// TIA Portal project "FillerMachine" (V15)
// Maquina llenadora Fuente Pura CCN

(* hardware
DEVICE "ET 200SP station_1"  ET 200SP-Station
   slot 0: "Rack_0"  Rack  6ES5 710-8MAx1
   slot 1: "PLC_1"  CPU 1510SP-1 PN  6ES7 510-1DJ01-0AB0  V2.5
   slot 2: "DI 8x24VDC ST_1"  DI 8x24VDC ST  6ES7 131-6BF00-0BA0  V1.1
      slot 1: "DI 8x24VDC ST_1"  DI 8x24VDC ST
   slot 3: "DI 8x24VDC ST_2"  DI 8x24VDC ST  6ES7 131-6BF01-0BA0  V0.0
      slot 1: "DI 8x24VDC ST_2"  DI 8x24VDC ST
   slot 4: "DI 8x24VDC ST_3"  DI 8x24VDC ST  6ES7 131-6BF01-0BA0  V0.0
      slot 1: "DI 8x24VDC ST_3"  DI 8x24VDC ST
   slot 5: "DQ 8x24VDC/0.5A ST_1"  DQ 8x24VDC/0.5A ST  6ES7 132-6BF01-0BA0  V0.0
      slot 1: "DQ 8x24VDC/0.5A ST_1"  DQ 8x24VDC/0.5A ST
   slot 6: "DQ 8x24VDC/0.5A ST_2"  DQ 8x24VDC/0.5A ST  6ES7 132-6BF01-0BA0  V0.0
      slot 1: "DQ 8x24VDC/0.5A ST_2"  DQ 8x24VDC/0.5A ST
   slot 7: "DQ 8x24VDC/0.5A ST_3"  DQ 8x24VDC/0.5A ST  6ES7 132-6BF01-0BA0  V0.0
      slot 1: "DQ 8x24VDC/0.5A ST_3"  DQ 8x24VDC/0.5A ST
   slot 8: "Server module_1"  Server module  6ES7 193-6PA00-0AA0  V1.1
      slot 1: "Server module_1"  Server module
   slot 127: "BA 2xRJ45"  BA 2xRJ45  6ES7 193-6AR00-0AA0  V0.0
      slot 32769: "Port_1"  6ES7 193-6AR00-0AA0
      slot 32770: "Port_2"  6ES7 193-6AR00-0AA0
DEVICE "HMI_1"  KTP600 Basic color PN
   slot 0: "HMI_1"  KTP600 Basic color PN  6AV6 647-0AD11-3AX0  12.0.0.0
   slot 1: "HMI_RT_2"  KTP600 Basic color PN  6AV6 647-0AD11-3AX0  12.0.0.0
   slot 5: "HMI_1.IE_CP_1"  PROFINET Interface  12.0.0.0
      slot 1: "PROFINET Interface_1"  PROFINET Interface
         slot 1: "Port_1"  Port
*)

// ===== PLC "PLC_1"  CPU 1510SP-1 PN =====

VAR_GLOBAL   // PLC tag table "Default tag table"
   "E_Stop" AT %I0.0 : Bool;
   "F_TriggerPump" AT %I0.1 : Bool;
   "ACKPump" AT %I0.2 : Bool;
   "F_TriggerClamp" AT %I0.3 : Bool;
   "ACKTap" AT %I0.4 : Bool;
   "F_TriggerTransp1" AT %I0.5 : Bool;
   "ACKTransp1" AT %I0.6 : Bool;
   "F_TriggerTransp2" AT %I0.7 : Bool;
   "ACKTransp2" AT %I1.0 : Bool;
   "S_ConvellorClearence_In" AT %I1.1 : Bool;
   "S_InBottle" AT %I1.2 : Bool;
   "S_OutBottle" AT %I1.6 : Bool;
   "S_LastBottle" AT %I1.4 : Bool;
   "S_Bottle_Convellor1" AT %I1.5 : Bool;
   "S_LevelH" AT %I1.3 : Bool;
   "S_LevelL" AT %I1.7 : Bool;
   "S_BottleTap" AT %I2.0 : Bool;
   "S_TranspClamp" AT %I2.1 : Bool;
   "PumpVLow" AT %Q0.0 : Bool;
   "PumpVHigh" AT %Q0.1 : Bool;
   "PumpStop" AT %Q0.2 : Bool;
   "MotorTap" AT %Q0.3 : Bool;
   "MotorTrans1" AT %Q0.4 : Bool;
   "MotorTrans2" AT %Q0.5 : Bool;
   "EVPrincip" AT %Q1.6 : Bool;
   "EVBlowCylindIN" AT %Q1.7 : Bool;
   "EVCylindBottleHigh" AT %Q2.0 : Bool;
   "EVCylindNeck" AT %Q2.1 : Bool;
   "EVDoorIn" AT %Q2.2 : Bool;
   "EVDoorOut" AT %Q2.3 : Bool;
   "EVClampBotNeck" AT %Q2.4 : Bool;
   "EVClampDoor" AT %Q2.5 : Bool;
   "EVSuperClamp" AT %Q2.6 : Bool;
   "EVMandrilcylindUpDown" AT %Q2.7 : Bool;
   "Start_hmi" AT %M11.0 : Bool;
   "MBandaT-On" AT %M10.1 : Bool;
   "MFillScreen" AT %M10.2 : Bool;
   "MBottleProcess" AT %MD100 : DInt;
   "MBottleCounterIN" AT %MD108 : DInt;
   "MBottleCounterOut" AT %MD128 : DInt;
   "MEnableClampValve" AT %MD132 : DInt;
   "MFillFinish" AT %M10.3 : Bool;
   "M_stop_hmi" AT %M11.1 : Bool;
   "S_ConvellorClearence_bit" AT %M20.3 : Bool;
   "S_InBottle_bit" AT %M20.4 : Bool;
   "S_OutBottle_bit" AT %M20.5 : Bool;
   "S_LastBottle_bit" AT %M20.6 : Bool;
   "S_Bottle_Convellor1_bit" AT %M20.7 : Bool;
   "S_LevelH_bit" AT %M21.0 : Bool;
   "S_LevelL_bit" AT %M21.1 : Bool;
   "S_BottleTap_bit" AT %M21.2 : Bool;
   "S_TranspClamp_bit" AT %M21.3 : Bool;
   "PumpVLow_bit" AT %M21.4 : Bool;
   "PumpVHigh_bit" AT %M21.5 : Bool;
   "PumpStop_bit" AT %M21.6 : Bool;
   "MotorTap_bit" AT %M21.7 : Bool;
   "MotorTrans1_bit" AT %M22.0 : Bool;
   "MotorTrans2_bit" AT %M22.1 : Bool;
   "EVPrincip_bit" AT %M22.2 : Bool;
   "EVBlowCylindIN_bit" AT %M22.3 : Bool;
   "EVMandrilcylindUpDown_bit" AT %M22.4 : Bool;
   "EVCylindNeck_bit" AT %M22.5 : Bool;
   "EVDoorIn_bit" AT %M50.1 : Bool;
   "EVDoorOut_bit" AT %M22.7 : Bool;
   "EVClampBotNeck_bit" AT %M23.0 : Bool;
   "EVClampDoor_bit" AT %M23.1 : Bool;
   "EVSuperClamp_bit" AT %M23.2 : Bool;
   "Alarm" AT %M24.0 : Bool;
   "F_TriggerPump_bit" AT %M24.1 : Bool;
   "F_TriggerClamp_bit" AT %M24.3 : Bool;
   "F_TriggerTransp1_bit" AT %M24.5 : Bool;
   "F_TriggerTransp2_bit" AT %M24.7 : Bool;
   "Run" AT %M25.1 : Bool;
   "Stop_bit" AT %M25.2 : Bool;
   "StageLL0" AT %M25.3 : Bool;
   "StageLL1" AT %M25.4 : Bool;
   "MBottleCounterR" AT %M25.5 : Bool;
   "ProcessFillingTimeR" AT %M25.6 : Bool;
   "StageLL2" AT %M25.7 : Bool;
   "MBottleclampRt" AT %M27.3 : Bool;
   "E_Trans1_hmi" AT %M27.4 : Bool;
   "E_Trans2_hmi" AT %M27.5 : Bool;
   "Pump_hmi" AT %M27.6 : Bool;
   "E_MotorTap_hmi" AT %M27.7 : Bool;
   "EVCylindBottleHigh_bit" AT %M28.0 : Bool;
   "StageLL3" AT %M28.1 : Bool;
   "StageLL4" AT %M28.2 : Bool;
   "StageLL5" AT %M28.3 : Bool;
   "StageLL6" AT %M28.4 : Bool;
   "StageLL7" AT %M28.5 : Bool;
   "StageLL8" AT %M28.6 : Bool;
   "StageLL9" AT %M28.7 : Bool;
   "StageLL10" AT %M29.0 : Bool;
   "StageLL11" AT %M29.1 : Bool;
   "Tag_1" AT %M400.1 : Bool;
   "StageLL12" AT %M29.2 : Bool;
   "StageLL13" AT %M29.3 : Bool;
   "StageLL14" AT %M29.4 : Bool;
   "Tag_2" AT %M400.2 : Bool;
   "StageLL00" AT %M29.5 : Bool;
   "MBottleCounterOutR" AT %M29.6 : Bool;
   "StageTap0" AT %M29.7 : Bool;
   "StageTap1" AT %M30.0 : Bool;
   "StageTap2" AT %M30.1 : Bool;
   "StageTap3" AT %M30.2 : Bool;
   "StageTap4" AT %M30.3 : Bool;
   "StageTap5" AT %M30.4 : Bool;
   "MTapProcessR" AT %M30.5 : Bool;
   "StageCon0" AT %M30.6 : Bool;
   "StageCon1" AT %M30.7 : Bool;
   "StageCon2" AT %M31.0 : Bool;
   "StageCon3" AT %M31.1 : Bool;
   "Timer1R" AT %M31.2 : Bool;
   "MConvT2R" AT %M31.3 : Bool;
   "StageCon4" AT %M31.4 : Bool;
   "E_stop_bit" AT %M31.5 : Bool;
   "ACKTap_bit" AT %M32.0 : Bool;
   "ACKPump_bit" AT %M32.1 : Bool;
   "ACKTransp1_bit" AT %M32.2 : Bool;
   "ACKTransp2_bit" AT %M32.3 : Bool;
   "MotorTap_fail" AT %M32.4 : Bool;
   "System_Byte" AT %MB1 : Byte;
   "RebuildMachine" AT %M1.0 : Bool;
   "DiagStatusUpdate" AT %M1.1 : Bool;
   "AlwaysTRUE" AT %M1.2 : Bool;
   "AlwaysFALSE" AT %M1.3 : Bool;
   "Clock_Byte" AT %MB0 : Byte;
   "Clock_10Hz" AT %M0.0 : Bool;
   "Clock_5Hz" AT %M0.1 : Bool;
   "Clock_2.5Hz" AT %M0.2 : Bool;
   "Clock_2Hz" AT %M0.3 : Bool;
   "Clock_1.25Hz" AT %M0.4 : Bool;
   "Clock_1Hz" AT %M0.5 : Bool;
   "Clock_0.625Hz" AT %M0.6 : Bool;
   "Clock_0.5Hz" AT %M0.7 : Bool;
   "MotorTransp1_fail" AT %M32.5 : Bool;
   "MotorTransp2_fail" AT %M32.6 : Bool;
   "MotorPump_fail" AT %M32.7 : Bool;
   "E_Manual" AT %M33.0 : Bool;
   "TimeFilling_hmi" AT %MD124 : Real;
   "TimeFilling_high" AT %MD104 : Real;
   "TimeFilling_low" AT %MD112 : Real;
   "TimeFilling_highT" AT %MD116 : Time;
   "TimeFilling_lowT" AT %MD120 : Time;
   "TimeFilling_highD" AT %MD54 : DInt;
   "TimeFilling_lowD" AT %MD58 : DInt;
   "TimeFilling_highPer" AT %MD62 : Real;
   "TimeFilling_lowPer" AT %MD66 : Real;
   "M_Stop" AT %M37.2 : Bool;
   "M_Stop_Counter_R" AT %M37.0 : Bool;
   "Stop_Batch" AT %M37.1 : Bool;
   "TapPPM" AT %MW4 : Word;
   "ResetTapPPM" AT %M37.3 : Bool;
   "ONS1" AT %M37.4 : Bool;
   "TapPPM_HMI" AT %MW6 : Word;
   "EstimatePPM_HMI" AT %MD70 : Real;
   "PumpVLow_hmi" AT %M37.5 : Bool;
   "EVBlowCylindIN_hmi" AT %M37.6 : Bool;
   "EVCylindBottleHigh_hmi" AT %M37.7 : Bool;
   "EVCylindNeck_hmi" AT %M39.0 : Bool;
   "EVPrincip_hmi" AT %M39.1 : Bool;
   "EVDoorIn_hmi" AT %M50.0 : Bool;
   "EVDoorOut_hmi" AT %M39.3 : Bool;
   "EVClampBotNeck_hmi" AT %M39.4 : Bool;
   "EVClampDoor_hmi" AT %M39.5 : Bool;
   "EVSuperClamp_hmi" AT %M50.2 : Bool;
   "EVMandrilcylindUpDown_hmi" AT %M50.3 : Bool;
   "E_Manual_hmi" AT %M31.6 : Bool;
   "Tag_3" AT %I2.4 : Bool;
   "Tag_4" AT %I2.3 : Bool;
   "Tag_5" AT %M24.2 : Bool;
   "Tag_6" AT %M140.1 : Bool;
   "Tag_7" AT %MD150 : DInt;
   "Tag_8" AT %MD154 : DInt;
   "Tag_9" AT %MD158 : DInt;
   "Tag_10" AT %MD162 : DInt;
   "Tag_11" AT %MD166 : DInt;
   "Tag_12" AT %MD170 : DInt;
   "Tag_13" AT %MD172 : DInt;
   "Tag_14" AT %MD176 : DInt;
   "Tag_15" AT %MD180 : DInt;
   "Tag_16" AT %MD184 : DInt;
   "Tag_17" AT %MD188 : Real;
   "Tag_18" AT %MD192 : Real;
   "Tag_19" AT %MD200 : Real;
   "Tag_20" AT %MD204 : Real;
   "Tag_21" AT %MD208 : Real;
   "Tag_22" AT %MD212 : Real;
   "Tag_23" AT %MD216 : Real;
   "Tag_24" AT %MD220 : Real;
   "Tag_25" AT %MD224 : Real;
   "Tag_26" AT %MD228 : Real;
   "Tag_27" AT %MD232 : Real;
   "Tag_28" AT %MD236 : Real;
   "R_time_b_neck" AT %M40.0 : Bool;
   "P_sensor_out" AT %M40.1 : Bool;
   "Tag_30" AT %MD240 : Real;
   "Tag_31" AT %MD244 : DInt;
   "PumpVHihg_hmi" AT %M40.2 : Bool;
   "Tag_32" AT %MD248 : Real;
   "Tag_33" AT %MD252 : DInt;
   "Tag_34" AT %MD256 : Real;
   "Tag_35" AT %MD260 : DInt;
   "P_Stop_hmi" AT %M40.4 : Bool;
   "Stop_hmi" AT %M40.5 : Bool;
   "WashProcess_1" AT %M10.4 : Bool;
   "WashProcess_hmi" AT %M10.5 : Bool;
   "RunWash" AT %M10.6 : Bool;
   "RWashProcess" AT %M10.7 : Bool;
   "Tag_36" AT %MD264 : Real;
   "Tag_37" AT %MD268 : DInt;
   "ValueProduction" AT %MD272 : DWord;
   "RProduction" AT %M31.7 : Bool;
   "Tag_29" AT %MD276 : Real;
   "Tag_38" AT %MD280 : DInt;
   "WashProcess_2" AT %M11.3 : Bool;
   "WashProcess_3" AT %M11.4 : Bool;
   "WashProcess_0" AT %M11.5 : Bool;
   "WashProcess_4" AT %M11.6 : Bool;
   "ret_val_RD_LOC" AT %MW284 : Int;
   "ret_val_RD_SYS" AT %MW288 : Int;
   "ret_val_WR_SYS" AT %MW292 : Int;
   "write_time" AT %M140.2 : Bool;
   "write_time_p" AT %M140.3 : Bool;
   "RestValve" AT %Q0.6 : Bool;
   "RestValve_bit" AT %M140.4 : Bool;
END_VAR

DATA_BLOCK "MotorTap_DB"   // DB1
{ S7_Optimized_Access := 'TRUE' }
VERSION : 0.1
// stored: InstanceOfName MotorData
"MotorData"
BEGIN
END_DATA_BLOCK

DATA_BLOCK "MotorTransp1_DB"   // DB5
{ S7_Optimized_Access := 'TRUE' }
VERSION : 0.1
// stored: InstanceOfName MotorData
"MotorData"
BEGIN
END_DATA_BLOCK

DATA_BLOCK "MotorTransp1"   // DB7
{ S7_Optimized_Access := 'TRUE' }
VERSION : 0.1
// stored: InstanceOfName MotorData
"MotorData"
BEGIN
END_DATA_BLOCK

DATA_BLOCK "MotorTransp2_DB"   // DB8
{ S7_Optimized_Access := 'TRUE' }
VERSION : 0.1
// stored: InstanceOfName MotorData
"MotorData"
BEGIN
END_DATA_BLOCK

DATA_BLOCK "init_var"   // DB9
{ S7_Optimized_Access := 'TRUE' }
VERSION : 0.1
   VAR RETAIN
      fillNo : Int := 8;
      filltime : Real := 9.0;
      fillPerHigh : Real := 70.0;
      fillPerLow : Real := 30.0;
   END_VAR
   VAR
      TimeConveyorBatch : Time := T#8.0S;
      TimeBeforeCylNeck : Time := T#0.5S;
      TimeCylNeck : Time := T#2S;
      TimeCylBottleHigh : Time := T#2S;
      TimeResetVLow : Time := T#2S;
      TimeRCyl_Neck_BottleHigh : Time := T#2S;
      TimeLastBottleOut : Time := T#2S;
      TimeClamp_Door_Neck : Time := T#2S;
      TimeClamp_Mandril : Time := T#2S;
      TimeSuperClamp : Time := T#0.05S;
   END_VAR
   VAR RETAIN
      RTimeConveyorBatch : Real := 2.0;
      RTimeBeforeCylNeck : Real := 0.5;
      RTimeCylBottleHigh : Real := 0.5;
      RTimeResetVLow : Real := 0.5;
      RTimeClamp_Door_Neck : Real := 0.5;
      RTimeClamp_Mandril : Real := 0.04;
      RTimeCylNeck : Real := 0.5;
      RTimeSuperClamp : Real := 2.0;
      RTimeRCyl_Neck_BottleHigh : Real := 1.0;
      RTimeRMandril_SuperClamp : Real := 2.0;
      RTimeLastBottleOut : Real := 0.5;
   END_VAR
   VAR
      TimeRMandril_SuperClamp : Time;
      TimeBNeck : Time;
   END_VAR
   VAR RETAIN
      RTimeBNeck : Real := 0.15;
      ROnDelayCylIn : Real := 0.5;
   END_VAR
   VAR
      TOnDelayCylIn : Time := T#0.5S;
   END_VAR
   VAR RETAIN
      ROnDelayDoorIn : Real := 0.9;
   END_VAR
   VAR
      TOnDelayDoorIn : Time := T#0.9S;
   END_VAR
   VAR RETAIN
      ROnDelayNeckClamp : Real := 0.5;
   END_VAR
   VAR
      TOnDelayNeckClamp : Time := T#0.5S;
      TWashTime : Time := T#120S;
   END_VAR
   VAR RETAIN
      RWashTime : Real := 120.0;
   END_VAR
BEGIN
END_DATA_BLOCK

DATA_BLOCK "DB_Alarms"   // DB13
{ S7_Optimized_Access := 'FALSE' }
VERSION : 0.1
   VAR
      E_Stop_alm : Bool;
      T_Pump_alm : Bool;
      T_Transp1_alm : Bool;
      T_Transp2_alm : Bool;
      T_Clamp_alm_1 : Bool;
      alarms_active : Bool;
   END_VAR
BEGIN
END_DATA_BLOCK

DATA_BLOCK "DB_Time"   // DB19
{ S7_Optimized_Access := 'TRUE' }
VERSION : 0.1
   VAR
      time_local_Read : DTL;
      time_system_WRITE : DTL;
   END_VAR
BEGIN
END_DATA_BLOCK

// folder: System blocks/Program resources

DATA_BLOCK "TimerStage2"   // DB2
{ S7_Optimized_Access := 'TRUE' }
AUTHOR : Simatic
FAMILY : IEC
NAME : IEC_TMR
VERSION : 1.0
// stored: InstanceOfName IEC_TIMER
"IEC_TIMER"
BEGIN
END_DATA_BLOCK

DATA_BLOCK "Timer_Cyl_Out"   // DB3
{ S7_Optimized_Access := 'TRUE' }
AUTHOR : Simatic
FAMILY : IEC
NAME : IEC_TMR
VERSION : 1.0
// stored: InstanceOfName IEC_TIMER
"IEC_TIMER"
BEGIN
END_DATA_BLOCK

DATA_BLOCK "TimeNeckWash"   // DB4
{ S7_Optimized_Access := 'TRUE' }
AUTHOR : Simatic
FAMILY : IEC
NAME : IEC_TMR
VERSION : 1.0
// stored: InstanceOfName IEC_TIMER
"IEC_TIMER"
BEGIN
END_DATA_BLOCK

DATA_BLOCK "IEC_Timer_0_DB_4"   // DB6
{ S7_Optimized_Access := 'TRUE' }
AUTHOR : Simatic
FAMILY : IEC
NAME : IEC_TMR
VERSION : 1.0
// stored: InstanceOfName IEC_TIMER
"IEC_TIMER"
BEGIN
END_DATA_BLOCK

DATA_BLOCK "CounterTapPPM"   // DB10
{ S7_Optimized_Access := 'TRUE' }
AUTHOR : Simatic
FAMILY : IEC
NAME : CNTR
VERSION : 1.0
// stored: InstanceOfName IEC_COUNTER
"IEC_COUNTER"
BEGIN
END_DATA_BLOCK

DATA_BLOCK "CounterTap"   // DB11
{ S7_Optimized_Access := 'TRUE' }
AUTHOR : Simatic
FAMILY : IEC
NAME : CNTR
VERSION : 1.0
// stored: InstanceOfName IEC_COUNTER
"IEC_COUNTER"
BEGIN
END_DATA_BLOCK

DATA_BLOCK "Delay_door_in"   // DB12
{ S7_Optimized_Access := 'TRUE' }
AUTHOR : Simatic
FAMILY : IEC
NAME : IEC_TMR
VERSION : 1.0
// stored: InstanceOfName IEC_TIMER
"IEC_TIMER"
BEGIN
END_DATA_BLOCK

DATA_BLOCK "TimerPPMDisable"   // DB14
{ S7_Optimized_Access := 'TRUE' }
AUTHOR : Simatic
FAMILY : IEC
NAME : IEC_TMR
VERSION : 1.0
// stored: InstanceOfName IEC_TIMER
"IEC_TIMER"
BEGIN
END_DATA_BLOCK

DATA_BLOCK "IEC_Timer_0_DB"   // DB15
{ S7_Optimized_Access := 'TRUE' }
AUTHOR : Simatic
FAMILY : IEC
NAME : IEC_TMR
VERSION : 1.0
// stored: InstanceOfName IEC_TIMER
"IEC_TIMER"
BEGIN
END_DATA_BLOCK

DATA_BLOCK "TimerStageWash"   // DB16
{ S7_Optimized_Access := 'TRUE' }
AUTHOR : Simatic
FAMILY : IEC
NAME : IEC_TMR
VERSION : 1.0
// stored: InstanceOfName IEC_TIMER
"IEC_TIMER"
BEGIN
END_DATA_BLOCK

DATA_BLOCK "TimeValvWash"   // DB17
{ S7_Optimized_Access := 'TRUE' }
AUTHOR : Simatic
FAMILY : IEC
NAME : IEC_TMR
VERSION : 1.0
// stored: InstanceOfName IEC_TIMER
"IEC_TIMER"
BEGIN
END_DATA_BLOCK

DATA_BLOCK "CounterProduction"   // DB18
{ S7_Optimized_Access := 'TRUE' }
AUTHOR : Simatic
FAMILY : IEC
NAME : CNTR
VERSION : 1.0
// stored: InstanceOfName IEC_COUNTER
"IEC_COUNTER"
BEGIN
END_DATA_BLOCK

DATA_BLOCK "TimerStage3"   // DB21
{ S7_Optimized_Access := 'TRUE' }
AUTHOR : Simatic
FAMILY : IEC
NAME : IEC_TMR
VERSION : 1.0
// stored: InstanceOfName IEC_TIMER
"IEC_TIMER"
BEGIN
END_DATA_BLOCK

DATA_BLOCK "TimerStage4"   // DB22
{ S7_Optimized_Access := 'TRUE' }
AUTHOR : Simatic
FAMILY : IEC
NAME : IEC_TMR
VERSION : 1.0
// stored: InstanceOfName IEC_TIMER
"IEC_TIMER"
BEGIN
END_DATA_BLOCK

DATA_BLOCK "TimerStage5"   // DB23
{ S7_Optimized_Access := 'TRUE' }
AUTHOR : Simatic
FAMILY : IEC
NAME : IEC_TMR
VERSION : 1.0
// stored: InstanceOfName IEC_TIMER
"IEC_TIMER"
BEGIN
END_DATA_BLOCK

DATA_BLOCK "TimerStage6"   // DB24
{ S7_Optimized_Access := 'TRUE' }
AUTHOR : Simatic
FAMILY : IEC
NAME : IEC_TMR
VERSION : 1.0
// stored: InstanceOfName IEC_TIMER
"IEC_TIMER"
BEGIN
END_DATA_BLOCK

DATA_BLOCK "TimerStage7"   // DB25
{ S7_Optimized_Access := 'TRUE' }
AUTHOR : Simatic
FAMILY : IEC
NAME : IEC_TMR
VERSION : 1.0
// stored: InstanceOfName IEC_TIMER
"IEC_TIMER"
BEGIN
END_DATA_BLOCK

DATA_BLOCK "TimerStage8"   // DB26
{ S7_Optimized_Access := 'TRUE' }
AUTHOR : Simatic
FAMILY : IEC
NAME : IEC_TMR
VERSION : 1.0
// stored: InstanceOfName IEC_TIMER
"IEC_TIMER"
BEGIN
END_DATA_BLOCK

DATA_BLOCK "CounterOut"   // DB27
{ S7_Optimized_Access := 'TRUE' }
AUTHOR : Simatic
FAMILY : IEC
NAME : CNTR
VERSION : 1.0
// stored: InstanceOfName IEC_COUNTER
"IEC_COUNTER"
BEGIN
END_DATA_BLOCK

DATA_BLOCK "TimerStageTap1"   // DB29
{ S7_Optimized_Access := 'TRUE' }
AUTHOR : Simatic
FAMILY : IEC
NAME : IEC_TMR
VERSION : 1.0
// stored: InstanceOfName IEC_TIMER
"IEC_TIMER"
BEGIN
END_DATA_BLOCK

DATA_BLOCK "TimerStageTap2"   // DB30
{ S7_Optimized_Access := 'TRUE' }
AUTHOR : Simatic
FAMILY : IEC
NAME : IEC_TMR
VERSION : 1.0
// stored: InstanceOfName IEC_TIMER
"IEC_TIMER"
BEGIN
END_DATA_BLOCK

DATA_BLOCK "TimerStageTap3"   // DB31
{ S7_Optimized_Access := 'TRUE' }
AUTHOR : Simatic
FAMILY : IEC
NAME : IEC_TMR
VERSION : 1.0
// stored: InstanceOfName IEC_TIMER
"IEC_TIMER"
BEGIN
END_DATA_BLOCK

DATA_BLOCK "TimerStageTap4"   // DB32
{ S7_Optimized_Access := 'TRUE' }
AUTHOR : Simatic
FAMILY : IEC
NAME : IEC_TMR
VERSION : 1.0
// stored: InstanceOfName IEC_TIMER
"IEC_TIMER"
BEGIN
END_DATA_BLOCK

DATA_BLOCK "TOnDelayStageCon2"   // DB33
{ S7_Optimized_Access := 'TRUE' }
AUTHOR : Simatic
FAMILY : IEC
NAME : IEC_TMR
VERSION : 1.0
// stored: InstanceOfName IEC_TIMER
"IEC_TIMER"
BEGIN
END_DATA_BLOCK

DATA_BLOCK "CounterIn"   // DB34
{ S7_Optimized_Access := 'TRUE' }
AUTHOR : Simatic
FAMILY : IEC
NAME : CNTR
VERSION : 1.0
// stored: InstanceOfName IEC_COUNTER
"IEC_COUNTER"
BEGIN
END_DATA_BLOCK

// folder: (top level)

FUNCTION_BLOCK "MotorData"   // FB1, LAD
{ S7_Optimized_Access := 'TRUE' }
VERSION : 0.1
   VAR_INPUT
      Ack_Motor : Bool;
      Alarms : Bool;
      Auto : Bool;
      Manual : Bool;
      Start : Bool;
   END_VAR
   VAR_OUTPUT
      Alarm_out : Bool;
   END_VAR
   VAR
      hrs : Real;
      Run : Bool;
      TimeMotor : DInt;
      TimeMotorE : Bool;
      clock : Bool;
      tag0 : Bool;
   END_VAR
   VAR RETAIN
      r_hrs : Real;
      min : DInt;
   END_VAR
   VAR
      IEC_Timer_0_Instance : TON_TIME;
   END_VAR
   VAR_TEMP   // added for the SCL form of the ladder/FBD networks
      _w1 : Bool;
   END_VAR
BEGIN

REGION Network 1
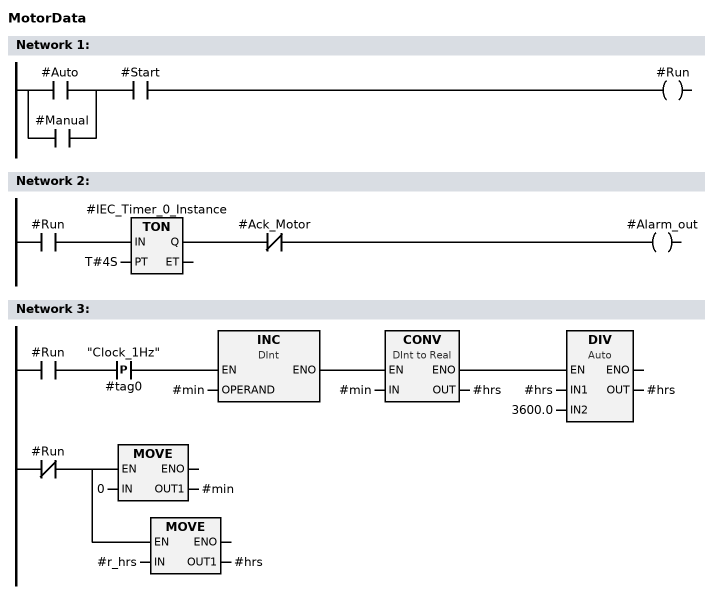
   RUNG wire#powerrail
      Contact( #Auto )
      wire#w1
      Contact( #Start )
      Coil( #Run )
   END_RUNG
   RUNG wire#powerrail
      Contact( #Manual )
   END_RUNG wire#w1
   // the same network as SCL:
   #Run := (#Auto OR #Manual) AND #Start;
END_REGION

REGION Network 2
   #IEC_Timer_0_Instance(IN := #Run, PT := T#4S);   // TON
   #Alarm_out := #IEC_Timer_0_Instance.Q AND NOT #Ack_Motor;
END_REGION

REGION Network 3
   RUNG wire#powerrail
      Contact( #Run )
      P_Contact(operand := "Clock_1Hz", bit := #tag0)
      { S7_Templates := "DestType := DInt" } Inc( #min )
      { S7_Templates := "[SrcType := DInt, DestType := Real]" } Convert(in := #min, out => #hrs)
      Div(in1 := #hrs, in2 := 3600.0, out => #hrs)
   END_RUNG
   RUNG wire#powerrail
      I_Contact( #Run )
      wire#w1
      Move(in := 0, out1 => #min)
   END_RUNG
   RUNG wire#w1
      Move(in := #r_hrs, out1 => #hrs)
   END_RUNG
   // the same network as SCL:
   #_w1 := #Run AND "Clock_1Hz" AND NOT #tag0;   // rising edge of "Clock_1Hz"
   #tag0 := "Clock_1Hz";
   IF #_w1 THEN
       #min := #min + 1;
       #hrs := DINT_TO_REAL(#min);
       #hrs := #hrs / 3600.0;
   END_IF;
   IF NOT #Run THEN
       #min := 0;
       #hrs := #r_hrs;
   END_IF;
END_REGION
END_FUNCTION_BLOCK

FUNCTION "Motor" : Void   // FC1, LAD
{ S7_Optimized_Access := 'TRUE' }
VERSION : 0.1
   VAR_INPUT
      ack : Bool;
      Run_1 : Bool;
   END_VAR
   VAR_OUTPUT
      motor : Bool;
   END_VAR
   VAR_IN_OUT
      IEC_Timer_0_Instance : TON_TIME;
   END_VAR
   VAR_TEMP
      TimeMotorE : Bool;
   END_VAR
BEGIN

REGION Network 1
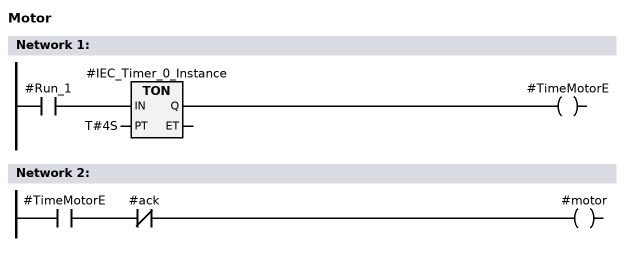
   #IEC_Timer_0_Instance(IN := #Run_1, PT := T#4S);   // TON
   #TimeMotorE := #IEC_Timer_0_Instance.Q;
END_REGION

REGION Network 2
   RUNG wire#powerrail
      Contact( #TimeMotorE )
      I_Contact( #ack )
      Coil( #motor )
   END_RUNG
   // the same network as SCL:
   #motor := #TimeMotorE AND NOT #ack;
END_REGION
END_FUNCTION

ORGANIZATION_BLOCK "Main"   // OB1, LAD, ProgramCycle
TITLE = "Main Program Sweep (Cycle)"
{ S7_Optimized_Access := 'TRUE' }
VERSION : 0.1
   VAR_INPUT
      Initial_Call : Bool;   // Initial call of this OB
      Remanence : Bool;   // =True, if remanent data are available
   END_VAR
   VAR_TEMP   // added for the SCL form of the ladder/FBD networks
      _w1 : Bool;
      _w2 : Bool;
   END_VAR
BEGIN

REGION Network 1
   // Start  Stop Control
   // Corregir Alarm a NC
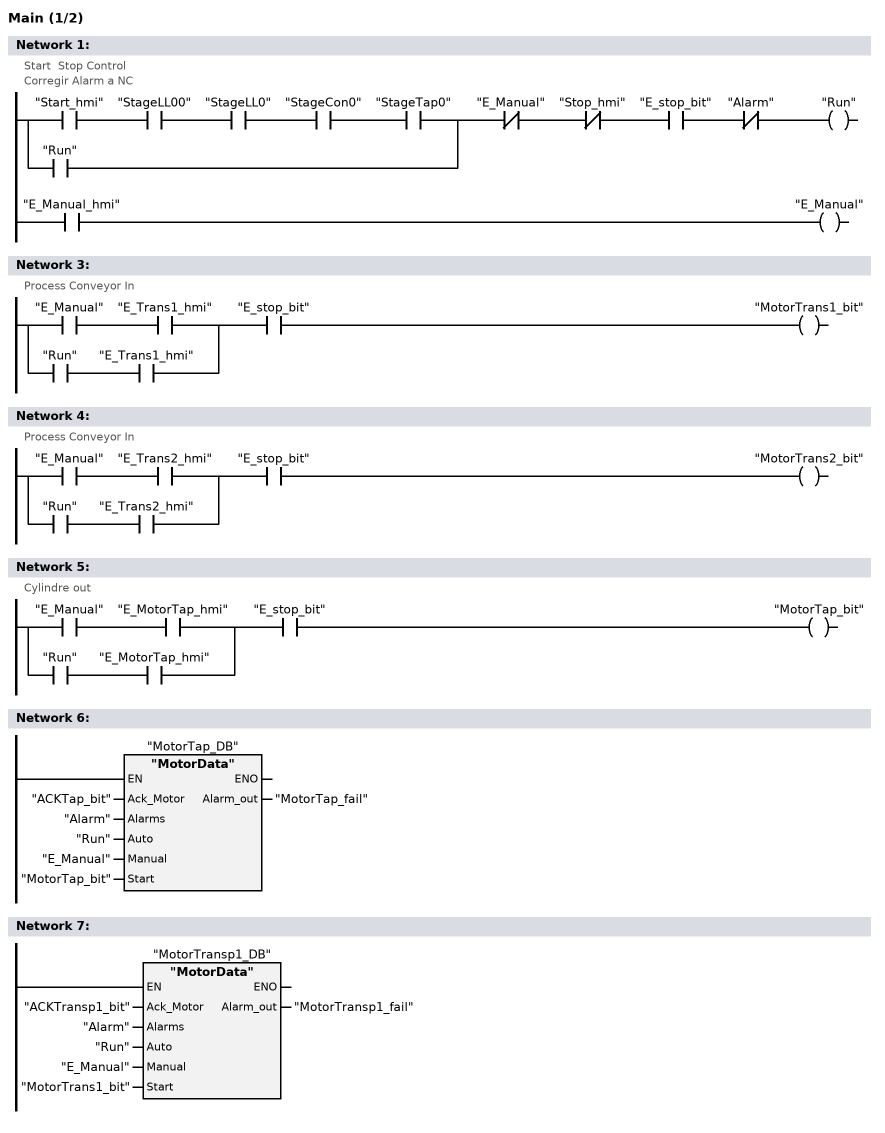
   RUNG wire#powerrail
      Contact( "Start_hmi" )
      Contact( "StageLL00" )
      Contact( "StageLL0" )
      Contact( "StageCon0" )
      Contact( "StageTap0" )
      wire#w1
      I_Contact( "E_Manual" )
      I_Contact( "Stop_hmi" )
      Contact( "E_stop_bit" )
      I_Contact( "Alarm" )
      Coil( "Run" )
   END_RUNG
   RUNG wire#powerrail
      Contact( "Run" )
   END_RUNG wire#w1
   RUNG wire#powerrail
      Contact( "E_Manual_hmi" )
      Coil( "E_Manual" )
   END_RUNG
   // the same network as SCL:
   "Run" := (("Start_hmi" AND "StageLL00" AND "StageLL0" AND "StageCon0" AND "StageTap0") OR "Run") AND NOT "E_Manual" AND NOT "Stop_hmi" AND "E_stop_bit" AND NOT "Alarm";
   "E_Manual" := "E_Manual_hmi";
END_REGION

REGION Network 2
   // Tank fill
END_REGION

REGION Network 3
   // Process Conveyor In
   RUNG wire#powerrail
      Contact( "E_Manual" )
      Contact( "E_Trans1_hmi" )
      wire#w1
      Contact( "E_stop_bit" )
      Coil( "MotorTrans1_bit" )
   END_RUNG
   RUNG wire#powerrail
      Contact( "Run" )
      Contact( "E_Trans1_hmi" )
   END_RUNG wire#w1
   // the same network as SCL:
   "MotorTrans1_bit" := (("E_Manual" AND "E_Trans1_hmi") OR ("Run" AND "E_Trans1_hmi")) AND "E_stop_bit";
END_REGION

REGION Network 4
   // Process Conveyor In
   RUNG wire#powerrail
      Contact( "E_Manual" )
      Contact( "E_Trans2_hmi" )
      wire#w1
      Contact( "E_stop_bit" )
      Coil( "MotorTrans2_bit" )
   END_RUNG
   RUNG wire#powerrail
      Contact( "Run" )
      Contact( "E_Trans2_hmi" )
   END_RUNG wire#w1
   // the same network as SCL:
   "MotorTrans2_bit" := (("E_Manual" AND "E_Trans2_hmi") OR ("Run" AND "E_Trans2_hmi")) AND "E_stop_bit";
END_REGION

REGION Network 5
   // Cylindre out
   RUNG wire#powerrail
      Contact( "E_Manual" )
      Contact( "E_MotorTap_hmi" )
      wire#w1
      Contact( "E_stop_bit" )
      Coil( "MotorTap_bit" )
   END_RUNG
   RUNG wire#powerrail
      Contact( "Run" )
      Contact( "E_MotorTap_hmi" )
   END_RUNG wire#w1
   // the same network as SCL:
   "MotorTap_bit" := (("E_Manual" AND "E_MotorTap_hmi") OR ("Run" AND "E_MotorTap_hmi")) AND "E_stop_bit";
END_REGION

REGION Network 6
   RUNG wire#powerrail
      "MotorTap_DB"(Ack_Motor := "ACKTap_bit", Alarms := "Alarm", Auto := "Run", Manual := "E_Manual", Start := "MotorTap_bit", Alarm_out => "MotorTap_fail")
   END_RUNG
   // the same network as SCL:
   "MotorTap_DB"(Ack_Motor := "ACKTap_bit",   // "MotorData"
                 Alarms := "Alarm",
                 Auto := "Run",
                 Manual := "E_Manual",
                 Start := "MotorTap_bit",
                 Alarm_out => "MotorTap_fail");
END_REGION

REGION Network 7
   RUNG wire#powerrail
      "MotorTransp1_DB"(Ack_Motor := "ACKTransp1_bit", Alarms := "Alarm", Auto := "Run", Manual := "E_Manual", Start := "MotorTrans1_bit", Alarm_out => "MotorTransp1_fail")
   END_RUNG
   // the same network as SCL:
   "MotorTransp1_DB"(Ack_Motor := "ACKTransp1_bit",   // "MotorData"
                     Alarms := "Alarm",
                     Auto := "Run",
                     Manual := "E_Manual",
                     Start := "MotorTrans1_bit",
                     Alarm_out => "MotorTransp1_fail");
END_REGION

REGION Network 8
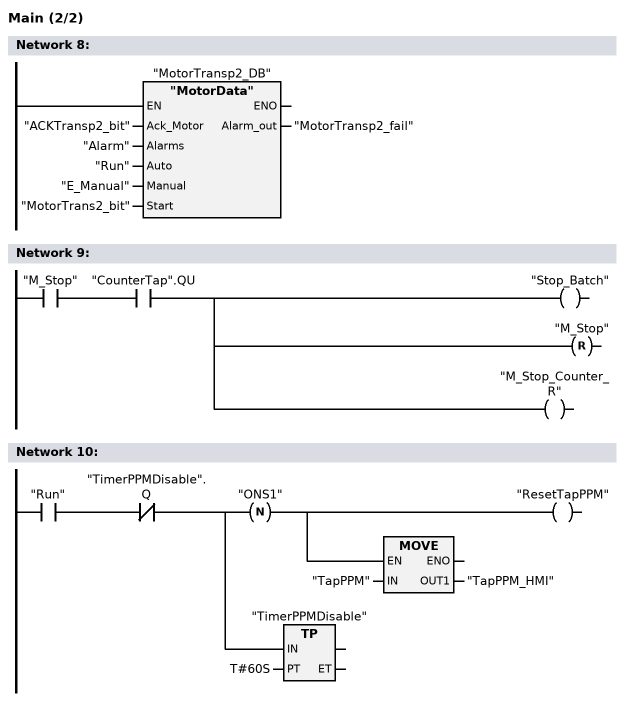
   RUNG wire#powerrail
      "MotorTransp2_DB"(Ack_Motor := "ACKTransp2_bit", Alarms := "Alarm", Auto := "Run", Manual := "E_Manual", Start := "MotorTrans2_bit", Alarm_out => "MotorTransp2_fail")
   END_RUNG
   // the same network as SCL:
   "MotorTransp2_DB"(Ack_Motor := "ACKTransp2_bit",   // "MotorData"
                     Alarms := "Alarm",
                     Auto := "Run",
                     Manual := "E_Manual",
                     Start := "MotorTrans2_bit",
                     Alarm_out => "MotorTransp2_fail");
END_REGION

REGION Network 9
   RUNG wire#powerrail
      Contact( "M_Stop" )
      Contact( "CounterTap".QU )
      wire#w1
      Coil( "Stop_Batch" )
   END_RUNG
   RUNG wire#w1
      R_Coil( "M_Stop" )
   END_RUNG
   RUNG wire#w1
      Coil( "M_Stop_Counter_R" )
   END_RUNG
   // the same network as SCL:
   "Stop_Batch" := "M_Stop" AND "CounterTap".QU;
   IF "Stop_Batch" THEN "M_Stop" := FALSE; END_IF;
   "M_Stop_Counter_R" := "Stop_Batch";
END_REGION

REGION Network 10
   #_w1 := "Run" AND NOT "TimerPPMDisable".Q;
   #_w2 := NOT #_w1 AND "ONS1";   // falling edge
   "ONS1" := #_w1;
   "ResetTapPPM" := #_w2;
   IF #_w2 THEN "TapPPM_HMI" := "TapPPM"; END_IF;
   "TimerPPMDisable".TP(IN := #_w1, PT := T#60S);
END_REGION
END_ORGANIZATION_BLOCK

ORGANIZATION_BLOCK "Alarms_block"   // OB123, LAD, ProgramCycle
TITLE = "Main Program Sweep (Cycle)"
{ S7_Optimized_Access := 'TRUE' }
VERSION : 0.1
   VAR_INPUT
      Initial_Call : Bool;   // Initial call of this OB
      Remanence : Bool;   // =True, if remanent data are available
   END_VAR
BEGIN

REGION Network 1
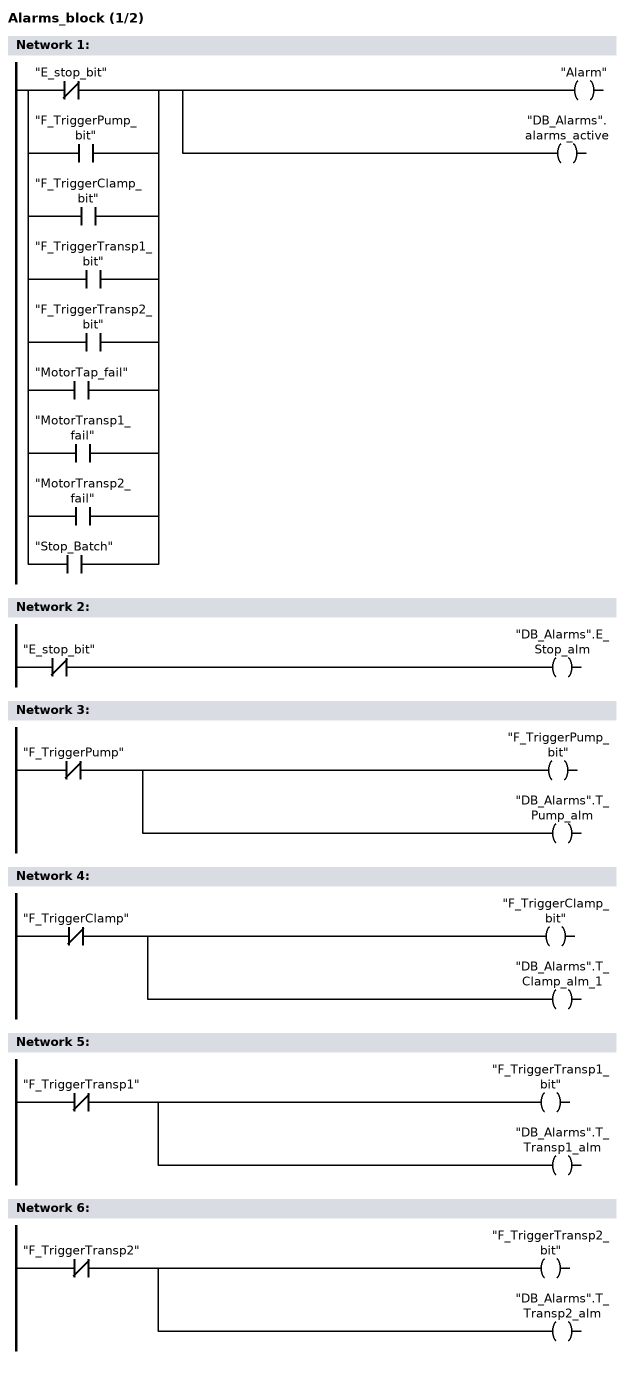
   RUNG wire#powerrail
      I_Contact( "E_stop_bit" )
      wire#w1
      Coil( "Alarm" )
   END_RUNG
   RUNG wire#powerrail
      Contact( "F_TriggerPump_bit" )
   END_RUNG wire#w1
   RUNG wire#powerrail
      Contact( "F_TriggerClamp_bit" )
   END_RUNG wire#w1
   RUNG wire#powerrail
      Contact( "F_TriggerTransp1_bit" )
   END_RUNG wire#w1
   RUNG wire#powerrail
      Contact( "F_TriggerTransp2_bit" )
   END_RUNG wire#w1
   RUNG wire#powerrail
      Contact( "MotorTap_fail" )
   END_RUNG wire#w1
   RUNG wire#powerrail
      Contact( "MotorTransp1_fail" )
   END_RUNG wire#w1
   RUNG wire#powerrail
      Contact( "MotorTransp2_fail" )
   END_RUNG wire#w1
   RUNG wire#powerrail
      Contact( "Stop_Batch" )
   END_RUNG wire#w1
   RUNG wire#w1
      Coil( "DB_Alarms".alarms_active )
   END_RUNG
   // the same network as SCL:
   "Alarm" := NOT "E_stop_bit" OR "F_TriggerPump_bit" OR "F_TriggerClamp_bit" OR "F_TriggerTransp1_bit" OR "F_TriggerTransp2_bit" OR "MotorTap_fail" OR "MotorTransp1_fail" OR "MotorTransp2_fail" OR "Stop_Batch";
   "DB_Alarms".alarms_active := "Alarm";
END_REGION

REGION Network 2
   RUNG wire#powerrail
      I_Contact( "E_stop_bit" )
      Coil( "DB_Alarms".E_Stop_alm )
   END_RUNG
   // the same network as SCL:
   "DB_Alarms".E_Stop_alm := NOT "E_stop_bit";
END_REGION

REGION Network 3
   RUNG wire#powerrail
      I_Contact( "F_TriggerPump" )
      wire#w1
      Coil( "F_TriggerPump_bit" )
   END_RUNG
   RUNG wire#w1
      Coil( "DB_Alarms".T_Pump_alm )
   END_RUNG
   // the same network as SCL:
   "F_TriggerPump_bit" := NOT "F_TriggerPump";
   "DB_Alarms".T_Pump_alm := NOT "F_TriggerPump";
END_REGION

REGION Network 4
   RUNG wire#powerrail
      I_Contact( "F_TriggerClamp" )
      wire#w1
      Coil( "F_TriggerClamp_bit" )
   END_RUNG
   RUNG wire#w1
      Coil( "DB_Alarms".T_Clamp_alm_1 )
   END_RUNG
   // the same network as SCL:
   "F_TriggerClamp_bit" := NOT "F_TriggerClamp";
   "DB_Alarms".T_Clamp_alm_1 := NOT "F_TriggerClamp";
END_REGION

REGION Network 5
   RUNG wire#powerrail
      I_Contact( "F_TriggerTransp1" )
      wire#w1
      Coil( "F_TriggerTransp1_bit" )
   END_RUNG
   RUNG wire#w1
      Coil( "DB_Alarms".T_Transp1_alm )
   END_RUNG
   // the same network as SCL:
   "F_TriggerTransp1_bit" := NOT "F_TriggerTransp1";
   "DB_Alarms".T_Transp1_alm := NOT "F_TriggerTransp1";
END_REGION

REGION Network 6
   RUNG wire#powerrail
      I_Contact( "F_TriggerTransp2" )
      wire#w1
      Coil( "F_TriggerTransp2_bit" )
   END_RUNG
   RUNG wire#w1
      Coil( "DB_Alarms".T_Transp2_alm )
   END_RUNG
   // the same network as SCL:
   "F_TriggerTransp2_bit" := NOT "F_TriggerTransp2";
   "DB_Alarms".T_Transp2_alm := NOT "F_TriggerTransp2";
END_REGION

REGION Network 7
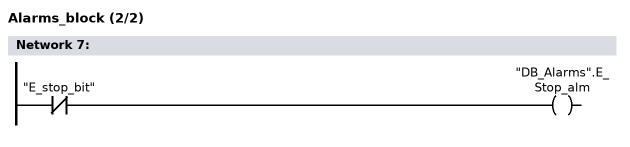
   RUNG wire#powerrail
      I_Contact( "E_stop_bit" )
      Coil( "DB_Alarms".E_Stop_alm )
   END_RUNG
   // the same network as SCL:
   "DB_Alarms".E_Stop_alm := NOT "E_stop_bit";
END_REGION
END_ORGANIZATION_BLOCK

ORGANIZATION_BLOCK "Stages"   // OB124, LAD, ProgramCycle
TITLE = "Main Program Sweep (Cycle)"
{ S7_Optimized_Access := 'TRUE' }
VERSION : 0.1
   VAR_INPUT
      Initial_Call : Bool;   // Initial call of this OB
      Remanence : Bool;   // =True, if remanent data are available
   END_VAR
   VAR_TEMP   // added for the SCL form of the ladder/FBD networks
      _w1 : Bool;
      _w2 : Bool;
      _w3 : Bool;
      _w4 : Bool;
      _w5 : Bool;
      _w6 : Bool;
      _w7 : Bool;
      _w8 : Bool;
      _w9 : Bool;
      _w10 : Bool;
   END_VAR
BEGIN

REGION Network 1
   // Stage0
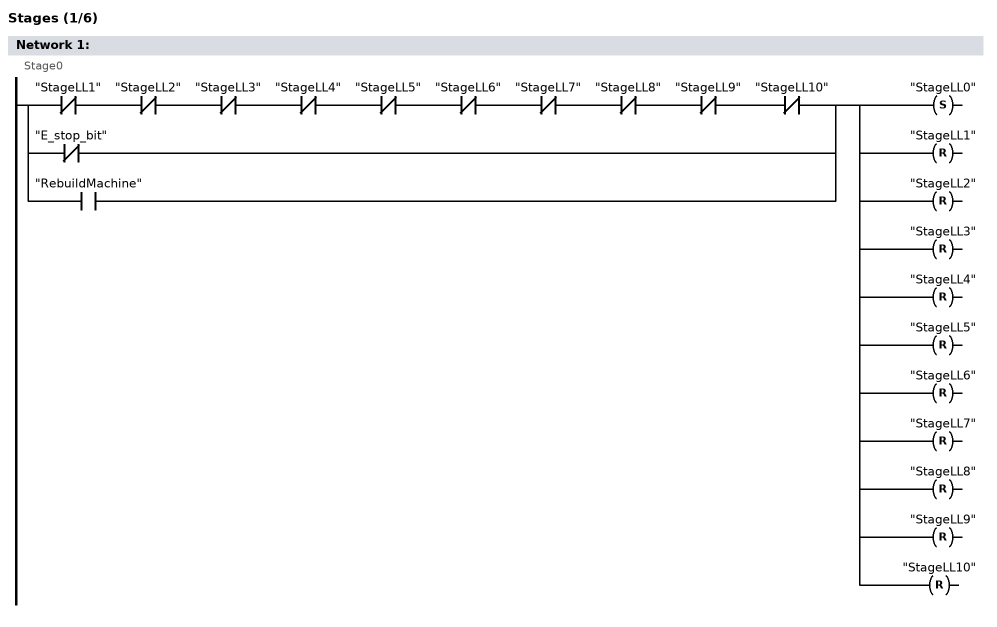
   RUNG wire#powerrail
      I_Contact( "StageLL1" )
      I_Contact( "StageLL2" )
      I_Contact( "StageLL3" )
      I_Contact( "StageLL4" )
      I_Contact( "StageLL5" )
      I_Contact( "StageLL6" )
      I_Contact( "StageLL7" )
      I_Contact( "StageLL8" )
      I_Contact( "StageLL9" )
      I_Contact( "StageLL10" )
      wire#w1
      S_Coil( "StageLL0" )
   END_RUNG
   RUNG wire#powerrail
      I_Contact( "E_stop_bit" )
   END_RUNG wire#w1
   RUNG wire#powerrail
      Contact( "RebuildMachine" )
   END_RUNG wire#w1
   RUNG wire#w1
      R_Coil( "StageLL1" )
   END_RUNG
   RUNG wire#w1
      R_Coil( "StageLL2" )
   END_RUNG
   RUNG wire#w1
      R_Coil( "StageLL3" )
   END_RUNG
   RUNG wire#w1
      R_Coil( "StageLL4" )
   END_RUNG
   RUNG wire#w1
      R_Coil( "StageLL5" )
   END_RUNG
   RUNG wire#w1
      R_Coil( "StageLL6" )
   END_RUNG
   RUNG wire#w1
      R_Coil( "StageLL7" )
   END_RUNG
   RUNG wire#w1
      R_Coil( "StageLL8" )
   END_RUNG
   RUNG wire#w1
      R_Coil( "StageLL9" )
   END_RUNG
   RUNG wire#w1
      R_Coil( "StageLL10" )
   END_RUNG
   // the same network as SCL:
   IF (NOT "StageLL1" AND NOT "StageLL2" AND NOT "StageLL3" AND NOT "StageLL4" AND NOT "StageLL5" AND NOT "StageLL6" AND NOT "StageLL7" AND NOT "StageLL8" AND NOT "StageLL9" AND NOT "StageLL10") OR NOT "E_stop_bit" OR "RebuildMachine" THEN
       "StageLL0" := TRUE;
   END_IF;
   #_w1 := (NOT "StageLL1" AND NOT "StageLL2" AND NOT "StageLL3" AND NOT "StageLL4" AND NOT "StageLL5" AND NOT "StageLL6" AND NOT "StageLL7" AND NOT "StageLL8" AND NOT "StageLL9" AND NOT "StageLL10") OR NOT "E_stop_bit" OR "RebuildMachine";
   IF #_w1 THEN
       "StageLL1" := FALSE;
       "StageLL2" := FALSE;
       "StageLL3" := FALSE;
       "StageLL4" := FALSE;
       "StageLL5" := FALSE;
       "StageLL6" := FALSE;
       "StageLL7" := FALSE;
       "StageLL8" := FALSE;
       "StageLL9" := FALSE;
       "StageLL10" := FALSE;
   END_IF;
END_REGION

REGION Network 2
   // ;LHGFEtapas de Cilindro de entrada y Llenado de Galones
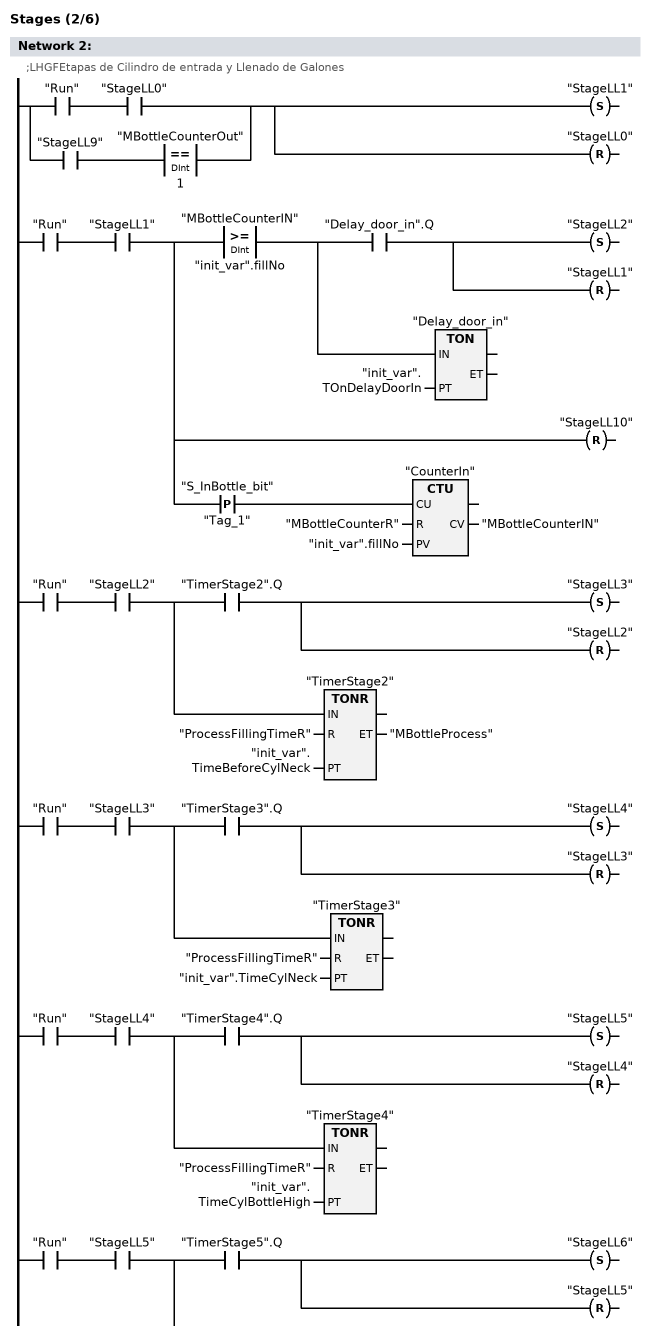
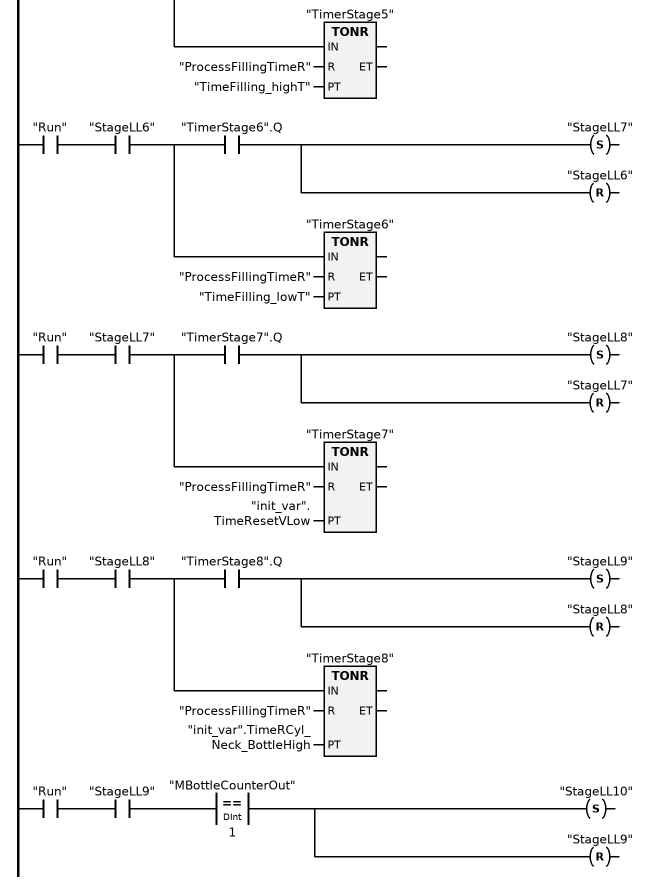
   IF ("Run" AND "StageLL0") OR ("StageLL9" AND ("MBottleCounterOut" = 1)) THEN
       "StageLL1" := TRUE;
       "StageLL0" := FALSE;
   END_IF;
   #_w1 := "Run" AND "StageLL1";
   #_w2 := #_w1 AND ("MBottleCounterIN" >= "init_var".fillNo);
   IF #_w2 AND "Delay_door_in".Q THEN
       "StageLL2" := TRUE;
       "StageLL1" := FALSE;
   END_IF;
   "Delay_door_in".TON(IN := #_w2, PT := "init_var".TOnDelayDoorIn);
   IF #_w1 THEN "StageLL10" := FALSE; END_IF;
   #_w3 := #_w1 AND "S_InBottle_bit" AND NOT "Tag_1";   // rising edge of "S_InBottle_bit"
   "Tag_1" := "S_InBottle_bit";
   "CounterIn".CTU(CU := #_w3, R := "MBottleCounterR", PV := "init_var".fillNo, CV => "MBottleCounterIN");
   #_w4 := "Run" AND "StageLL2";
   IF #_w4 AND "TimerStage2".Q THEN
       "StageLL3" := TRUE;
       "StageLL2" := FALSE;
   END_IF;
   "TimerStage2".TONR(IN := #_w4,
                      R := "ProcessFillingTimeR",
                      PT := "init_var".TimeBeforeCylNeck,
                      ET => "MBottleProcess");
   #_w5 := "Run" AND "StageLL3";
   IF #_w5 AND "TimerStage3".Q THEN
       "StageLL4" := TRUE;
       "StageLL3" := FALSE;
   END_IF;
   "TimerStage3".TONR(IN := #_w5, R := "ProcessFillingTimeR", PT := "init_var".TimeCylNeck);
   #_w6 := "Run" AND "StageLL4";
   IF #_w6 AND "TimerStage4".Q THEN
       "StageLL5" := TRUE;
       "StageLL4" := FALSE;
   END_IF;
   "TimerStage4".TONR(IN := #_w6, R := "ProcessFillingTimeR", PT := "init_var".TimeCylBottleHigh);
   #_w7 := "Run" AND "StageLL5";
   IF #_w7 AND "TimerStage5".Q THEN
       "StageLL6" := TRUE;
       "StageLL5" := FALSE;
   END_IF;
   "TimerStage5".TONR(IN := #_w7, R := "ProcessFillingTimeR", PT := "TimeFilling_highT");
   #_w8 := "Run" AND "StageLL6";
   IF #_w8 AND "TimerStage6".Q THEN
       "StageLL7" := TRUE;
       "StageLL6" := FALSE;
   END_IF;
   "TimerStage6".TONR(IN := #_w8, R := "ProcessFillingTimeR", PT := "TimeFilling_lowT");
   #_w9 := "Run" AND "StageLL7";
   IF #_w9 AND "TimerStage7".Q THEN
       "StageLL8" := TRUE;
       "StageLL7" := FALSE;
   END_IF;
   "TimerStage7".TONR(IN := #_w9, R := "ProcessFillingTimeR", PT := "init_var".TimeResetVLow);
   #_w10 := "Run" AND "StageLL8";
   IF #_w10 AND "TimerStage8".Q THEN
       "StageLL9" := TRUE;
       "StageLL8" := FALSE;
   END_IF;
   "TimerStage8".TONR(IN := #_w10, R := "ProcessFillingTimeR", PT := "init_var".TimeRCyl_Neck_BottleHigh);
   IF "Run" AND "StageLL9" AND ("MBottleCounterOut" = 1) THEN
       "StageLL10" := TRUE;
       "StageLL9" := FALSE;
   END_IF;
END_REGION

REGION Network 3
   // Etapas de Cilindro de Salida
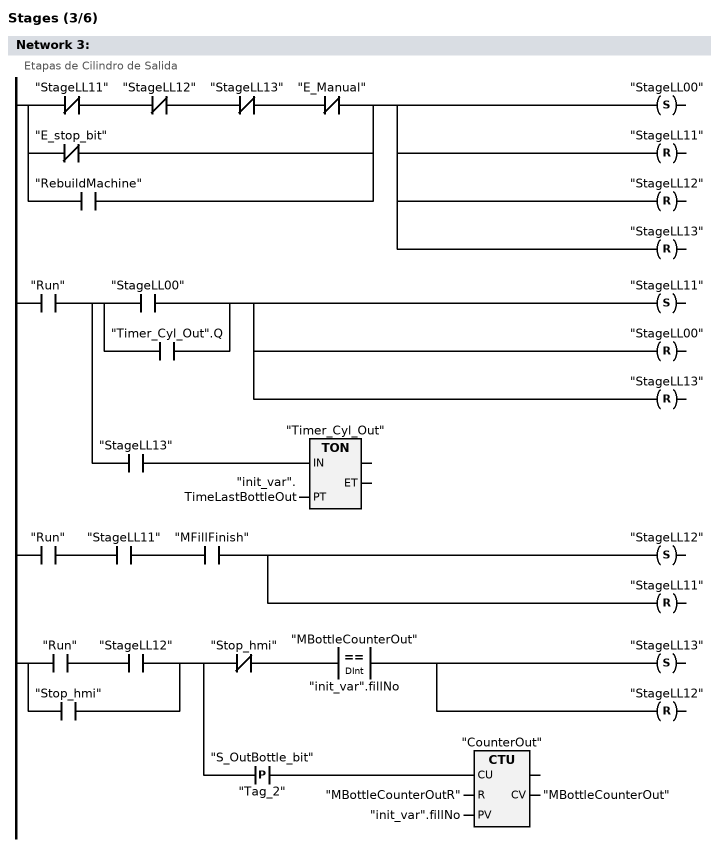
   IF (NOT "StageLL11" AND NOT "StageLL12" AND NOT "StageLL13" AND NOT "E_Manual") OR NOT "E_stop_bit" OR "RebuildMachine" THEN
       "StageLL00" := TRUE;
   END_IF;
   #_w1 := (NOT "StageLL11" AND NOT "StageLL12" AND NOT "StageLL13" AND NOT "E_Manual") OR NOT "E_stop_bit" OR "RebuildMachine";
   IF #_w1 THEN
       "StageLL11" := FALSE;
       "StageLL12" := FALSE;
       "StageLL13" := FALSE;
   END_IF;
   IF "Run" AND ("StageLL00" OR "Timer_Cyl_Out".Q) THEN "StageLL11" := TRUE; END_IF;
   #_w2 := "Run" AND ("StageLL00" OR "Timer_Cyl_Out".Q);
   IF #_w2 THEN
       "StageLL00" := FALSE;
       "StageLL13" := FALSE;
   END_IF;
   "Timer_Cyl_Out".TON(IN := "Run" AND "StageLL13", PT := "init_var".TimeLastBottleOut);
   IF "Run" AND "StageLL11" AND "MFillFinish" THEN
       "StageLL12" := TRUE;
       "StageLL11" := FALSE;
   END_IF;
   #_w3 := ("Run" AND "StageLL12") OR "Stop_hmi";
   IF #_w3 AND NOT "Stop_hmi" AND ("MBottleCounterOut" = "init_var".fillNo) THEN
       "StageLL13" := TRUE;
       "StageLL12" := FALSE;
   END_IF;
   #_w4 := #_w3 AND "S_OutBottle_bit" AND NOT "Tag_2";   // rising edge of "S_OutBottle_bit"
   "Tag_2" := "S_OutBottle_bit";
   "CounterOut".CTU(CU := #_w4, R := "MBottleCounterOutR", PV := "init_var".fillNo, CV => "MBottleCounterOut");
END_REGION

REGION Network 4
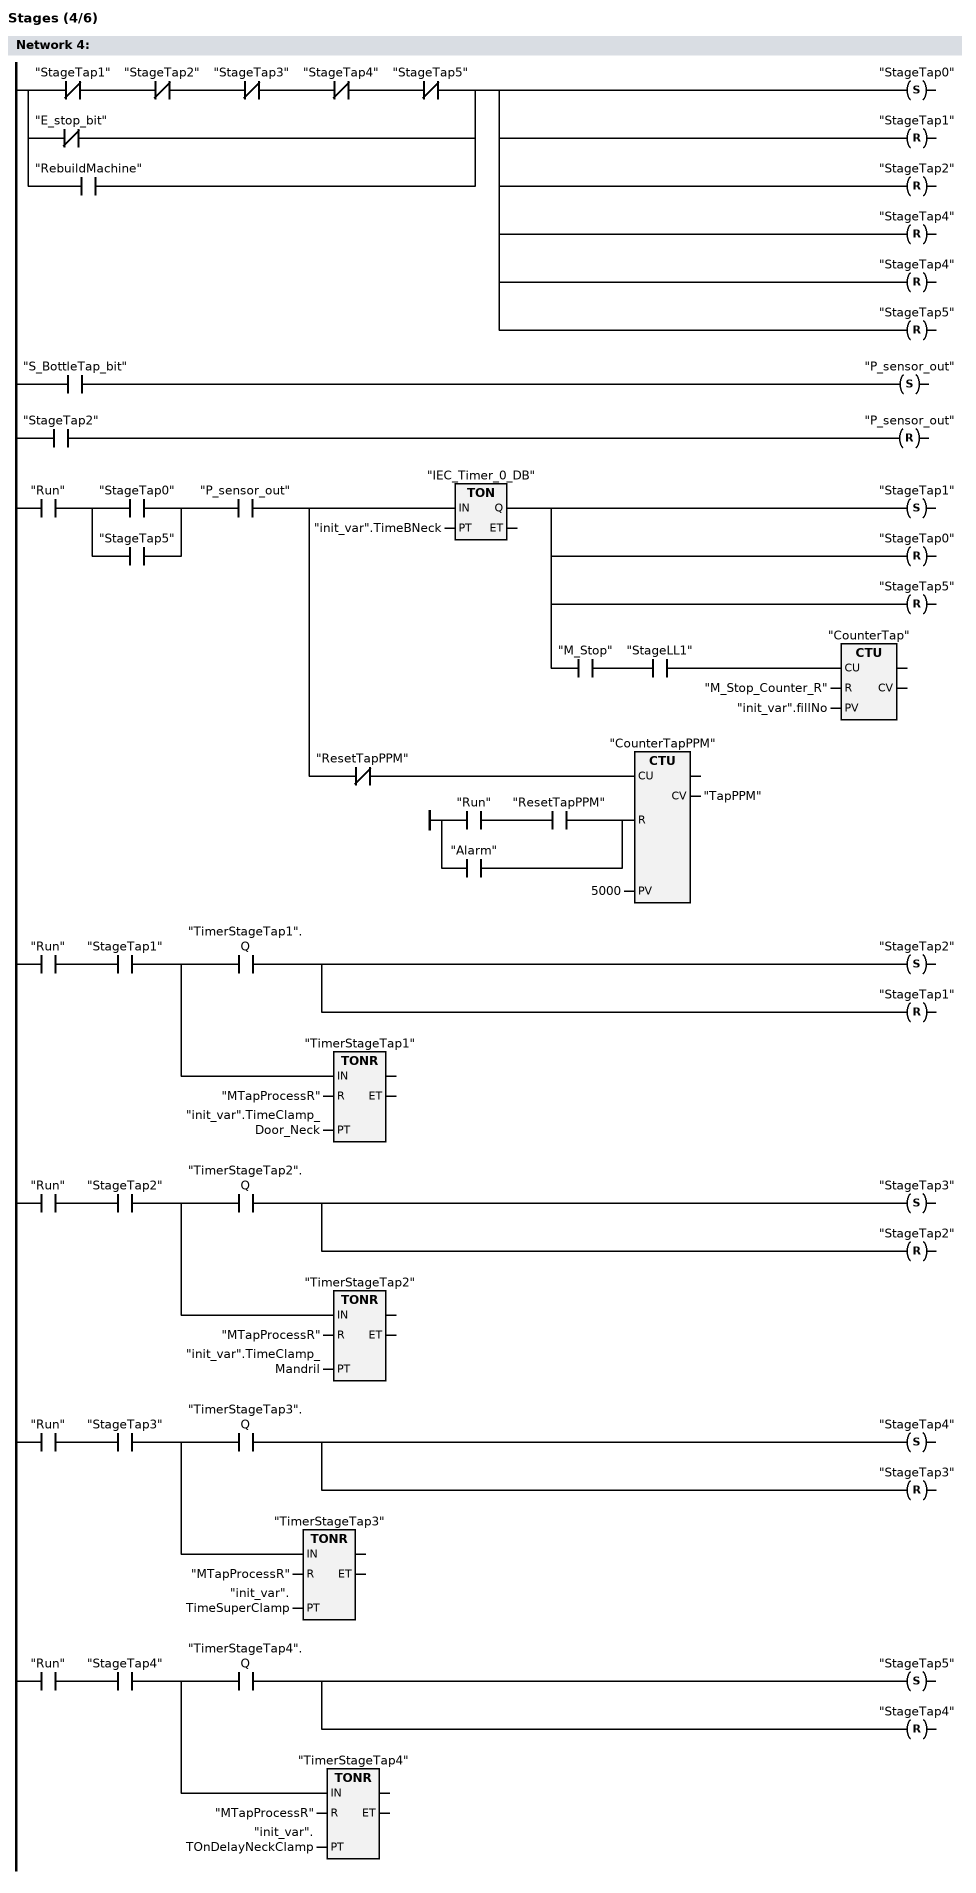
   IF (NOT "StageTap1" AND NOT "StageTap2" AND NOT "StageTap3" AND NOT "StageTap4" AND NOT "StageTap5") OR NOT "E_stop_bit" OR "RebuildMachine" THEN
       "StageTap0" := TRUE;
   END_IF;
   #_w1 := (NOT "StageTap1" AND NOT "StageTap2" AND NOT "StageTap3" AND NOT "StageTap4" AND NOT "StageTap5") OR NOT "E_stop_bit" OR "RebuildMachine";
   IF #_w1 THEN
       "StageTap1" := FALSE;
       "StageTap2" := FALSE;
       "StageTap4" := FALSE;
       "StageTap4" := FALSE;
       "StageTap5" := FALSE;
   END_IF;
   IF "S_BottleTap_bit" THEN "P_sensor_out" := TRUE; END_IF;
   IF "StageTap2" THEN "P_sensor_out" := FALSE; END_IF;
   #_w2 := "Run" AND ("StageTap0" OR "StageTap5") AND "P_sensor_out";
   "IEC_Timer_0_DB".TON(IN := #_w2, PT := "init_var".TimeBNeck);
   IF "IEC_Timer_0_DB".Q THEN
       "StageTap1" := TRUE;
       "StageTap0" := FALSE;
       "StageTap5" := FALSE;
   END_IF;
   "CounterTap".CTU(CU := "IEC_Timer_0_DB".Q AND "M_Stop" AND "StageLL1",
                    R := "M_Stop_Counter_R",
                    PV := "init_var".fillNo);
   "CounterTapPPM".CTU(CU := #_w2 AND NOT "ResetTapPPM",
                       R := ("Run" AND "ResetTapPPM") OR "Alarm",
                       PV := 5000,
                       CV => "TapPPM");
   #_w3 := "Run" AND "StageTap1";
   IF #_w3 AND "TimerStageTap1".Q THEN
       "StageTap2" := TRUE;
       "StageTap1" := FALSE;
   END_IF;
   "TimerStageTap1".TONR(IN := #_w3, R := "MTapProcessR", PT := "init_var".TimeClamp_Door_Neck);
   #_w4 := "Run" AND "StageTap2";
   IF #_w4 AND "TimerStageTap2".Q THEN
       "StageTap3" := TRUE;
       "StageTap2" := FALSE;
   END_IF;
   "TimerStageTap2".TONR(IN := #_w4, R := "MTapProcessR", PT := "init_var".TimeClamp_Mandril);
   #_w5 := "Run" AND "StageTap3";
   IF #_w5 AND "TimerStageTap3".Q THEN
       "StageTap4" := TRUE;
       "StageTap3" := FALSE;
   END_IF;
   "TimerStageTap3".TONR(IN := #_w5, R := "MTapProcessR", PT := "init_var".TimeSuperClamp);
   #_w6 := "Run" AND "StageTap4";
   IF #_w6 AND "TimerStageTap4".Q THEN
       "StageTap5" := TRUE;
       "StageTap4" := FALSE;
   END_IF;
   "TimerStageTap4".TONR(IN := #_w6, R := "MTapProcessR", PT := "init_var".TOnDelayNeckClamp);
END_REGION

REGION Network 5
   // Etapas Cilindro de entrada
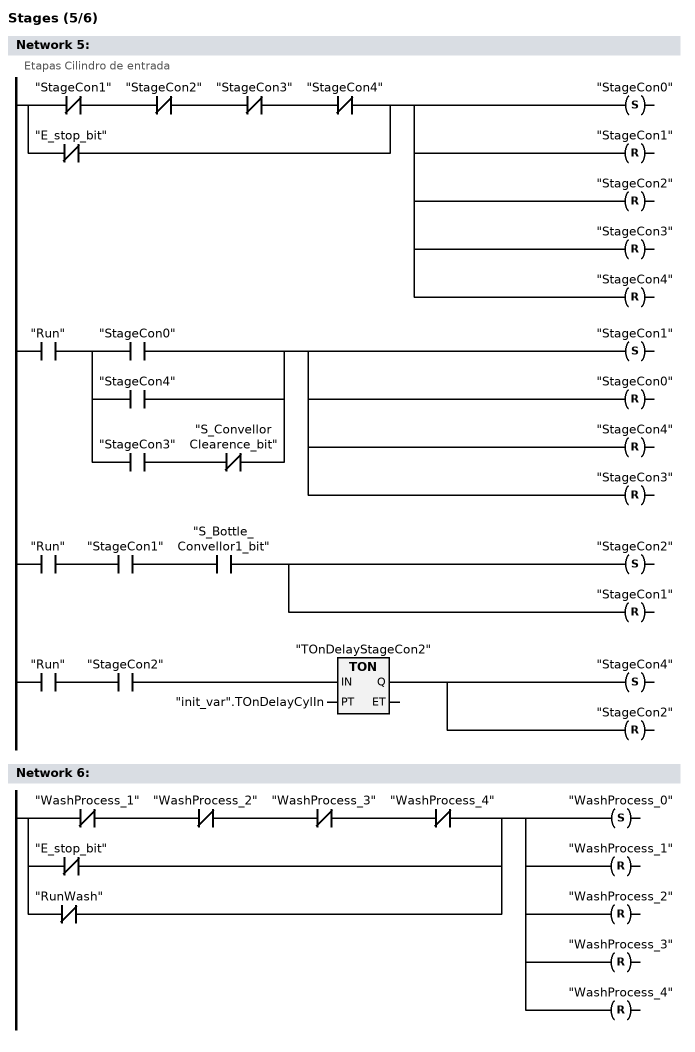
   IF (NOT "StageCon1" AND NOT "StageCon2" AND NOT "StageCon3" AND NOT "StageCon4") OR NOT "E_stop_bit" THEN
       "StageCon0" := TRUE;
   END_IF;
   #_w1 := (NOT "StageCon1" AND NOT "StageCon2" AND NOT "StageCon3" AND NOT "StageCon4") OR NOT "E_stop_bit";
   IF #_w1 THEN
       "StageCon1" := FALSE;
       "StageCon2" := FALSE;
       "StageCon3" := FALSE;
       "StageCon4" := FALSE;
   END_IF;
   IF "Run" AND ("StageCon0" OR "StageCon4" OR ("StageCon3" AND NOT "S_ConvellorClearence_bit")) THEN
       "StageCon1" := TRUE;
   END_IF;
   #_w2 := "Run" AND ("StageCon0" OR "StageCon4" OR ("StageCon3" AND NOT "S_ConvellorClearence_bit"));
   IF #_w2 THEN
       "StageCon0" := FALSE;
       "StageCon4" := FALSE;
       "StageCon3" := FALSE;
   END_IF;
   IF "Run" AND "StageCon1" AND "S_Bottle_Convellor1_bit" THEN
       "StageCon2" := TRUE;
       "StageCon1" := FALSE;
   END_IF;
   "TOnDelayStageCon2".TON(IN := "Run" AND "StageCon2", PT := "init_var".TOnDelayCylIn);
   IF "TOnDelayStageCon2".Q THEN
       "StageCon4" := TRUE;
       "StageCon2" := FALSE;
   END_IF;
END_REGION

REGION Network 6
   RUNG wire#powerrail
      I_Contact( "WashProcess_1" )
      I_Contact( "WashProcess_2" )
      I_Contact( "WashProcess_3" )
      I_Contact( "WashProcess_4" )
      wire#w1
      S_Coil( "WashProcess_0" )
   END_RUNG
   RUNG wire#powerrail
      I_Contact( "E_stop_bit" )
   END_RUNG wire#w1
   RUNG wire#powerrail
      I_Contact( "RunWash" )
   END_RUNG wire#w1
   RUNG wire#w1
      R_Coil( "WashProcess_1" )
   END_RUNG
   RUNG wire#w1
      R_Coil( "WashProcess_2" )
   END_RUNG
   RUNG wire#w1
      R_Coil( "WashProcess_3" )
   END_RUNG
   RUNG wire#w1
      R_Coil( "WashProcess_4" )
   END_RUNG
   // the same network as SCL:
   IF (NOT "WashProcess_1" AND NOT "WashProcess_2" AND NOT "WashProcess_3" AND NOT "WashProcess_4") OR NOT "E_stop_bit" OR NOT "RunWash" THEN
       "WashProcess_0" := TRUE;
   END_IF;
   #_w1 := (NOT "WashProcess_1" AND NOT "WashProcess_2" AND NOT "WashProcess_3" AND NOT "WashProcess_4") OR NOT "E_stop_bit" OR NOT "RunWash";
   IF #_w1 THEN
       "WashProcess_1" := FALSE;
       "WashProcess_2" := FALSE;
       "WashProcess_3" := FALSE;
       "WashProcess_4" := FALSE;
   END_IF;
END_REGION

REGION Network 7
   // Process Wash machine
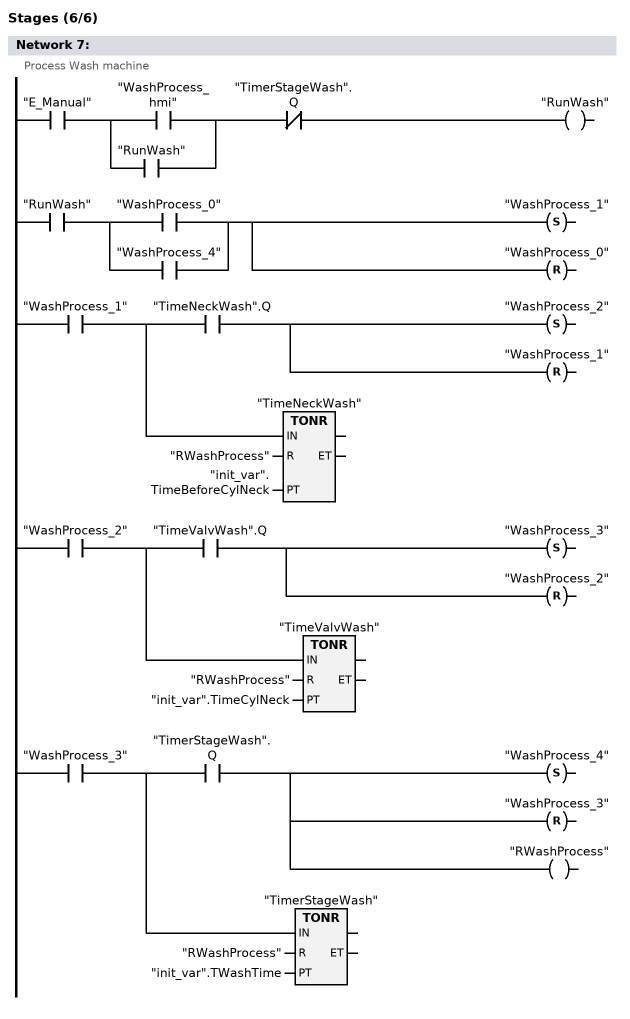
   "RunWash" := "E_Manual" AND ("WashProcess_hmi" OR "RunWash") AND NOT "TimerStageWash".Q;
   IF "RunWash" AND ("WashProcess_0" OR "WashProcess_4") THEN
       "WashProcess_1" := TRUE;
       "WashProcess_0" := FALSE;
   END_IF;
   IF "WashProcess_1" AND "TimeNeckWash".Q THEN "WashProcess_2" := TRUE; END_IF;
   #_w1 := "WashProcess_1";
   IF "WashProcess_1" AND "TimeNeckWash".Q THEN "WashProcess_1" := FALSE; END_IF;
   "TimeNeckWash".TONR(IN := #_w1, R := "RWashProcess", PT := "init_var".TimeBeforeCylNeck);
   IF "WashProcess_2" AND "TimeValvWash".Q THEN "WashProcess_3" := TRUE; END_IF;
   #_w2 := "WashProcess_2";
   IF "WashProcess_2" AND "TimeValvWash".Q THEN "WashProcess_2" := FALSE; END_IF;
   "TimeValvWash".TONR(IN := #_w2, R := "RWashProcess", PT := "init_var".TimeCylNeck);
   #_w3 := "WashProcess_3" AND "TimerStageWash".Q;
   IF #_w3 THEN "WashProcess_4" := TRUE; END_IF;
   #_w4 := "WashProcess_3";
   IF #_w3 THEN "WashProcess_3" := FALSE; END_IF;
   "RWashProcess" := #_w3;
   "TimerStageWash".TONR(IN := #_w4, R := "RWashProcess", PT := "init_var".TWashTime);
END_REGION

REGION Network 8
   // Stop Stage
END_REGION
END_ORGANIZATION_BLOCK

ORGANIZATION_BLOCK "Mirror_bits"   // OB125, LAD, ProgramCycle
TITLE = "Main Program Sweep (Cycle)"
{ S7_Optimized_Access := 'TRUE' }
VERSION : 0.1
   VAR_INPUT
      Initial_Call : Bool;   // Initial call of this OB
      Remanence : Bool;   // =True, if remanent data are available
   END_VAR
BEGIN

REGION Network 1
   // Minor Bits
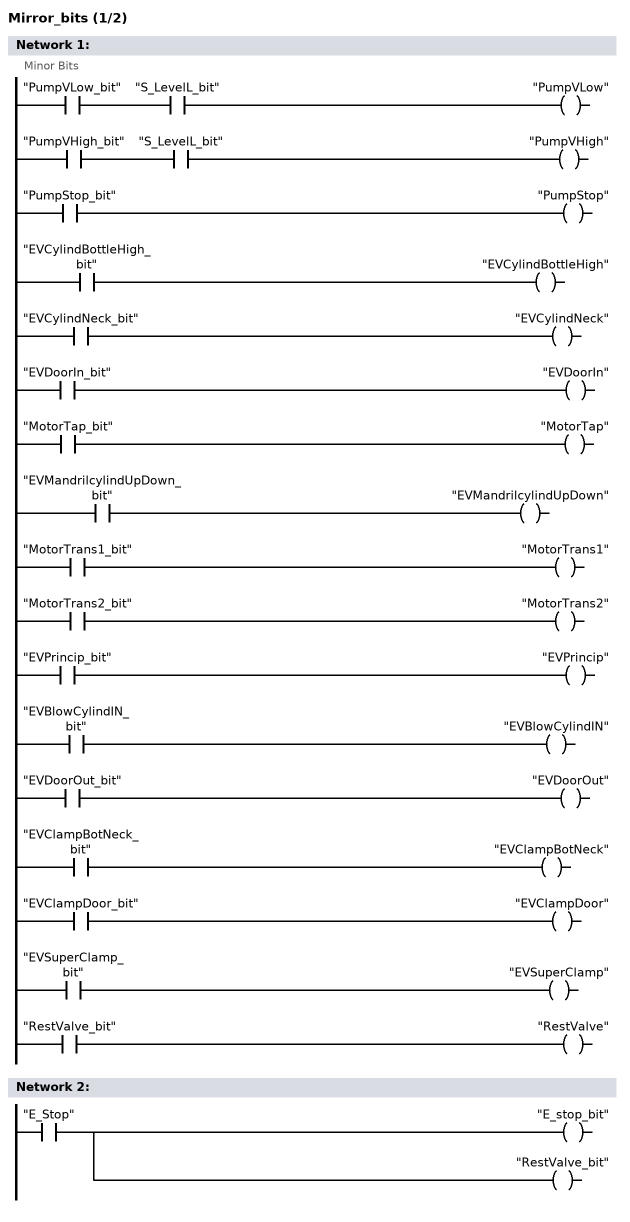
   RUNG wire#powerrail
      Contact( "PumpVLow_bit" )
      Contact( "S_LevelL_bit" )
      Coil( "PumpVLow" )
   END_RUNG
   RUNG wire#powerrail
      Contact( "PumpVHigh_bit" )
      Contact( "S_LevelL_bit" )
      Coil( "PumpVHigh" )
   END_RUNG
   RUNG wire#powerrail
      Contact( "PumpStop_bit" )
      Coil( "PumpStop" )
   END_RUNG
   RUNG wire#powerrail
      Contact( "EVCylindBottleHigh_bit" )
      Coil( "EVCylindBottleHigh" )
   END_RUNG
   RUNG wire#powerrail
      Contact( "EVCylindNeck_bit" )
      Coil( "EVCylindNeck" )
   END_RUNG
   RUNG wire#powerrail
      Contact( "EVDoorIn_bit" )
      Coil( "EVDoorIn" )
   END_RUNG
   RUNG wire#powerrail
      Contact( "MotorTap_bit" )
      Coil( "MotorTap" )
   END_RUNG
   RUNG wire#powerrail
      Contact( "EVMandrilcylindUpDown_bit" )
      Coil( "EVMandrilcylindUpDown" )
   END_RUNG
   RUNG wire#powerrail
      Contact( "MotorTrans1_bit" )
      Coil( "MotorTrans1" )
   END_RUNG
   RUNG wire#powerrail
      Contact( "MotorTrans2_bit" )
      Coil( "MotorTrans2" )
   END_RUNG
   RUNG wire#powerrail
      Contact( "EVPrincip_bit" )
      Coil( "EVPrincip" )
   END_RUNG
   RUNG wire#powerrail
      Contact( "EVBlowCylindIN_bit" )
      Coil( "EVBlowCylindIN" )
   END_RUNG
   RUNG wire#powerrail
      Contact( "EVDoorOut_bit" )
      Coil( "EVDoorOut" )
   END_RUNG
   RUNG wire#powerrail
      Contact( "EVClampBotNeck_bit" )
      Coil( "EVClampBotNeck" )
   END_RUNG
   RUNG wire#powerrail
      Contact( "EVClampDoor_bit" )
      Coil( "EVClampDoor" )
   END_RUNG
   RUNG wire#powerrail
      Contact( "EVSuperClamp_bit" )
      Coil( "EVSuperClamp" )
   END_RUNG
   RUNG wire#powerrail
      Contact( "RestValve_bit" )
      Coil( "RestValve" )
   END_RUNG
   // the same network as SCL:
   "PumpVLow" := "PumpVLow_bit" AND "S_LevelL_bit";
   "PumpVHigh" := "PumpVHigh_bit" AND "S_LevelL_bit";
   "PumpStop" := "PumpStop_bit";
   "EVCylindBottleHigh" := "EVCylindBottleHigh_bit";
   "EVCylindNeck" := "EVCylindNeck_bit";
   "EVDoorIn" := "EVDoorIn_bit";
   "MotorTap" := "MotorTap_bit";
   "EVMandrilcylindUpDown" := "EVMandrilcylindUpDown_bit";
   "MotorTrans1" := "MotorTrans1_bit";
   "MotorTrans2" := "MotorTrans2_bit";
   "EVPrincip" := "EVPrincip_bit";
   "EVBlowCylindIN" := "EVBlowCylindIN_bit";
   "EVDoorOut" := "EVDoorOut_bit";
   "EVClampBotNeck" := "EVClampBotNeck_bit";
   "EVClampDoor" := "EVClampDoor_bit";
   "EVSuperClamp" := "EVSuperClamp_bit";
   "RestValve" := "RestValve_bit";
END_REGION

REGION Network 2
   RUNG wire#powerrail
      Contact( "E_Stop" )
      wire#w1
      Coil( "E_stop_bit" )
   END_RUNG
   RUNG wire#w1
      Coil( "RestValve_bit" )
   END_RUNG
   // the same network as SCL:
   "E_stop_bit" := "E_Stop";
   "RestValve_bit" := "E_Stop";
END_REGION

REGION Network 3
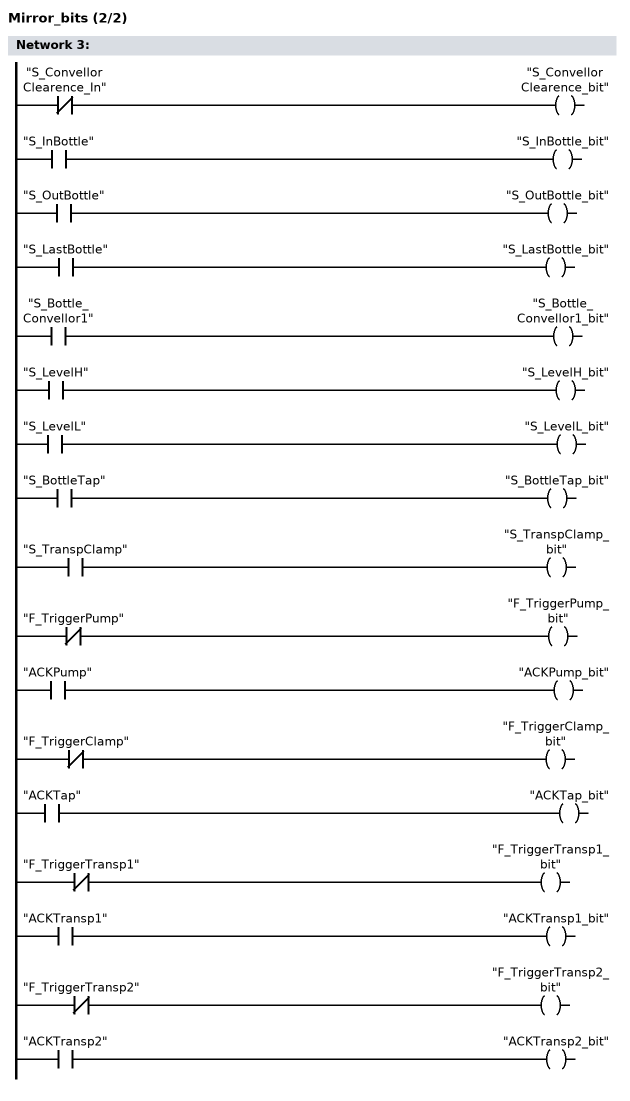
   RUNG wire#powerrail
      I_Contact( "S_ConvellorClearence_In" )
      Coil( "S_ConvellorClearence_bit" )
   END_RUNG
   RUNG wire#powerrail
      Contact( "S_InBottle" )
      Coil( "S_InBottle_bit" )
   END_RUNG
   RUNG wire#powerrail
      Contact( "S_OutBottle" )
      Coil( "S_OutBottle_bit" )
   END_RUNG
   RUNG wire#powerrail
      Contact( "S_LastBottle" )
      Coil( "S_LastBottle_bit" )
   END_RUNG
   RUNG wire#powerrail
      Contact( "S_Bottle_Convellor1" )
      Coil( "S_Bottle_Convellor1_bit" )
   END_RUNG
   RUNG wire#powerrail
      Contact( "S_LevelH" )
      Coil( "S_LevelH_bit" )
   END_RUNG
   RUNG wire#powerrail
      Contact( "S_LevelL" )
      Coil( "S_LevelL_bit" )
   END_RUNG
   RUNG wire#powerrail
      Contact( "S_BottleTap" )
      Coil( "S_BottleTap_bit" )
   END_RUNG
   RUNG wire#powerrail
      Contact( "S_TranspClamp" )
      Coil( "S_TranspClamp_bit" )
   END_RUNG
   RUNG wire#powerrail
      I_Contact( "F_TriggerPump" )
      Coil( "F_TriggerPump_bit" )
   END_RUNG
   RUNG wire#powerrail
      Contact( "ACKPump" )
      Coil( "ACKPump_bit" )
   END_RUNG
   RUNG wire#powerrail
      I_Contact( "F_TriggerClamp" )
      Coil( "F_TriggerClamp_bit" )
   END_RUNG
   RUNG wire#powerrail
      Contact( "ACKTap" )
      Coil( "ACKTap_bit" )
   END_RUNG
   RUNG wire#powerrail
      I_Contact( "F_TriggerTransp1" )
      Coil( "F_TriggerTransp1_bit" )
   END_RUNG
   RUNG wire#powerrail
      Contact( "ACKTransp1" )
      Coil( "ACKTransp1_bit" )
   END_RUNG
   RUNG wire#powerrail
      I_Contact( "F_TriggerTransp2" )
      Coil( "F_TriggerTransp2_bit" )
   END_RUNG
   RUNG wire#powerrail
      Contact( "ACKTransp2" )
      Coil( "ACKTransp2_bit" )
   END_RUNG
   // the same network as SCL:
   "S_ConvellorClearence_bit" := NOT "S_ConvellorClearence_In";
   "S_InBottle_bit" := "S_InBottle";
   "S_OutBottle_bit" := "S_OutBottle";
   "S_LastBottle_bit" := "S_LastBottle";
   "S_Bottle_Convellor1_bit" := "S_Bottle_Convellor1";
   "S_LevelH_bit" := "S_LevelH";
   "S_LevelL_bit" := "S_LevelL";
   "S_BottleTap_bit" := "S_BottleTap";
   "S_TranspClamp_bit" := "S_TranspClamp";
   "F_TriggerPump_bit" := NOT "F_TriggerPump";
   "ACKPump_bit" := "ACKPump";
   "F_TriggerClamp_bit" := NOT "F_TriggerClamp";
   "ACKTap_bit" := "ACKTap";
   "F_TriggerTransp1_bit" := NOT "F_TriggerTransp1";
   "ACKTransp1_bit" := "ACKTransp1";
   "F_TriggerTransp2_bit" := NOT "F_TriggerTransp2";
   "ACKTransp2_bit" := "ACKTransp2";
END_REGION
END_ORGANIZATION_BLOCK

ORGANIZATION_BLOCK "Actions"   // OB126, LAD, ProgramCycle
TITLE = "Main Program Sweep (Cycle)"
{ S7_Optimized_Access := 'TRUE' }
VERSION : 0.1
   VAR_INPUT
      Initial_Call : Bool;   // Initial call of this OB
      Remanence : Bool;   // =True, if remanent data are available
   END_VAR
BEGIN

REGION Network 1
   // VFD pin DCM (PumpStop_bit) enable, voltage source to pin VLow and VHigh
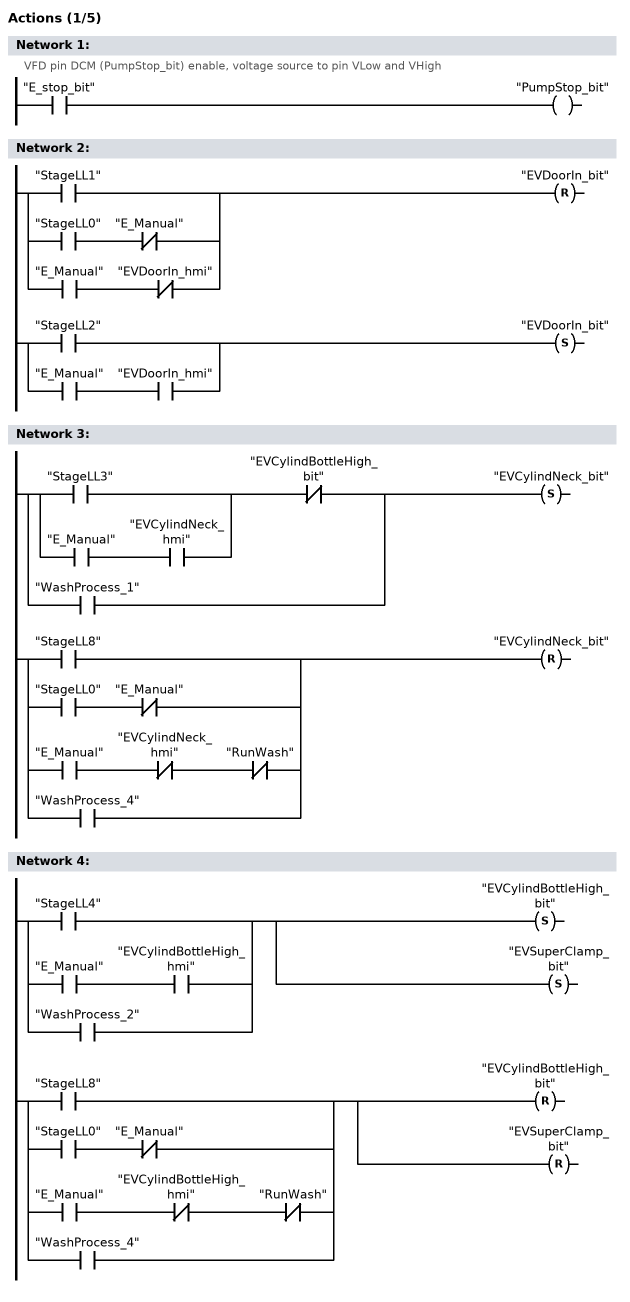
   RUNG wire#powerrail
      Contact( "E_stop_bit" )
      Coil( "PumpStop_bit" )
   END_RUNG
   // the same network as SCL:
   "PumpStop_bit" := "E_stop_bit";
END_REGION

REGION Network 2
   RUNG wire#powerrail
      Contact( "StageLL1" )
      wire#w1
      R_Coil( "EVDoorIn_bit" )
   END_RUNG
   RUNG wire#powerrail
      Contact( "StageLL0" )
      I_Contact( "E_Manual" )
   END_RUNG wire#w1
   RUNG wire#powerrail
      Contact( "E_Manual" )
      I_Contact( "EVDoorIn_hmi" )
   END_RUNG wire#w1
   RUNG wire#powerrail
      Contact( "StageLL2" )
      wire#w2
      S_Coil( "EVDoorIn_bit" )
   END_RUNG
   RUNG wire#powerrail
      Contact( "E_Manual" )
      Contact( "EVDoorIn_hmi" )
   END_RUNG wire#w2
   // the same network as SCL:
   IF "StageLL1" OR ("StageLL0" AND NOT "E_Manual") OR ("E_Manual" AND NOT "EVDoorIn_hmi") THEN
       "EVDoorIn_bit" := FALSE;
   END_IF;
   IF "StageLL2" OR ("E_Manual" AND "EVDoorIn_hmi") THEN "EVDoorIn_bit" := TRUE; END_IF;
END_REGION

REGION Network 3
   RUNG wire#powerrail
      Contact( "StageLL3" )
      wire#w1
      I_Contact( "EVCylindBottleHigh_bit" )
      wire#w2
      S_Coil( "EVCylindNeck_bit" )
   END_RUNG
   RUNG wire#powerrail
      Contact( "E_Manual" )
      Contact( "EVCylindNeck_hmi" )
   END_RUNG wire#w1
   RUNG wire#powerrail
      Contact( "WashProcess_1" )
   END_RUNG wire#w2
   RUNG wire#powerrail
      Contact( "StageLL8" )
      wire#w3
      R_Coil( "EVCylindNeck_bit" )
   END_RUNG
   RUNG wire#powerrail
      Contact( "StageLL0" )
      I_Contact( "E_Manual" )
   END_RUNG wire#w3
   RUNG wire#powerrail
      Contact( "E_Manual" )
      I_Contact( "EVCylindNeck_hmi" )
      I_Contact( "RunWash" )
   END_RUNG wire#w3
   RUNG wire#powerrail
      Contact( "WashProcess_4" )
   END_RUNG wire#w3
   // the same network as SCL:
   IF (("StageLL3" OR ("E_Manual" AND "EVCylindNeck_hmi")) AND NOT "EVCylindBottleHigh_bit") OR "WashProcess_1" THEN
       "EVCylindNeck_bit" := TRUE;
   END_IF;
   IF "StageLL8" OR ("StageLL0" AND NOT "E_Manual") OR ("E_Manual" AND NOT "EVCylindNeck_hmi" AND NOT "RunWash") OR "WashProcess_4" THEN
       "EVCylindNeck_bit" := FALSE;
   END_IF;
END_REGION

REGION Network 4
   RUNG wire#powerrail
      Contact( "StageLL4" )
      wire#w1
      S_Coil( "EVCylindBottleHigh_bit" )
   END_RUNG
   RUNG wire#powerrail
      Contact( "E_Manual" )
      Contact( "EVCylindBottleHigh_hmi" )
   END_RUNG wire#w1
   RUNG wire#powerrail
      Contact( "WashProcess_2" )
   END_RUNG wire#w1
   RUNG wire#w1
      S_Coil( "EVSuperClamp_bit" )
   END_RUNG
   RUNG wire#powerrail
      Contact( "StageLL8" )
      wire#w2
      R_Coil( "EVCylindBottleHigh_bit" )
   END_RUNG
   RUNG wire#powerrail
      Contact( "StageLL0" )
      I_Contact( "E_Manual" )
   END_RUNG wire#w2
   RUNG wire#powerrail
      Contact( "E_Manual" )
      I_Contact( "EVCylindBottleHigh_hmi" )
      I_Contact( "RunWash" )
   END_RUNG wire#w2
   RUNG wire#powerrail
      Contact( "WashProcess_4" )
   END_RUNG wire#w2
   RUNG wire#w2
      R_Coil( "EVSuperClamp_bit" )
   END_RUNG
   // the same network as SCL:
   IF "StageLL4" OR ("E_Manual" AND "EVCylindBottleHigh_hmi") OR "WashProcess_2" THEN
       "EVCylindBottleHigh_bit" := TRUE;
       "EVSuperClamp_bit" := TRUE;
   END_IF;
   IF "StageLL8" OR ("StageLL0" AND NOT "E_Manual") OR ("E_Manual" AND NOT "EVCylindBottleHigh_hmi" AND NOT "RunWash") OR "WashProcess_4" THEN
       "EVCylindBottleHigh_bit" := FALSE;
       "EVSuperClamp_bit" := FALSE;
   END_IF;
END_REGION

REGION Network 5
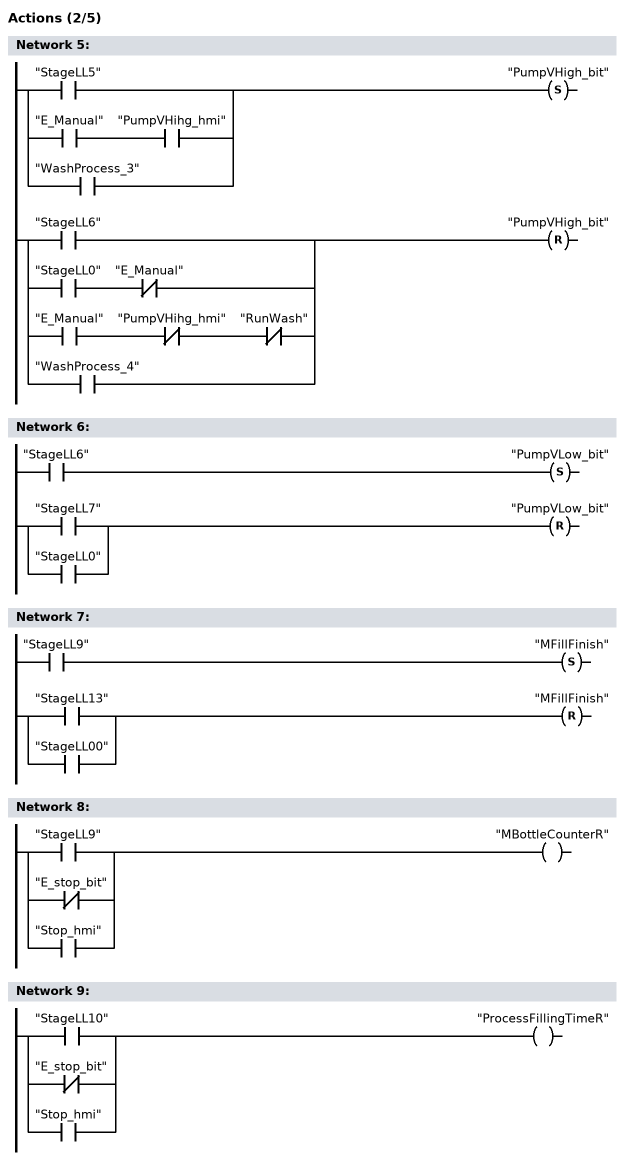
   RUNG wire#powerrail
      Contact( "StageLL5" )
      wire#w1
      S_Coil( "PumpVHigh_bit" )
   END_RUNG
   RUNG wire#powerrail
      Contact( "E_Manual" )
      Contact( "PumpVHihg_hmi" )
   END_RUNG wire#w1
   RUNG wire#powerrail
      Contact( "WashProcess_3" )
   END_RUNG wire#w1
   RUNG wire#powerrail
      Contact( "StageLL6" )
      wire#w2
      R_Coil( "PumpVHigh_bit" )
   END_RUNG
   RUNG wire#powerrail
      Contact( "StageLL0" )
      I_Contact( "E_Manual" )
   END_RUNG wire#w2
   RUNG wire#powerrail
      Contact( "E_Manual" )
      I_Contact( "PumpVHihg_hmi" )
      I_Contact( "RunWash" )
   END_RUNG wire#w2
   RUNG wire#powerrail
      Contact( "WashProcess_4" )
   END_RUNG wire#w2
   // the same network as SCL:
   IF "StageLL5" OR ("E_Manual" AND "PumpVHihg_hmi") OR "WashProcess_3" THEN "PumpVHigh_bit" := TRUE; END_IF;
   IF "StageLL6" OR ("StageLL0" AND NOT "E_Manual") OR ("E_Manual" AND NOT "PumpVHihg_hmi" AND NOT "RunWash") OR "WashProcess_4" THEN
       "PumpVHigh_bit" := FALSE;
   END_IF;
END_REGION

REGION Network 6
   RUNG wire#powerrail
      Contact( "StageLL6" )
      S_Coil( "PumpVLow_bit" )
   END_RUNG
   RUNG wire#powerrail
      Contact( "StageLL7" )
      wire#w1
      R_Coil( "PumpVLow_bit" )
   END_RUNG
   RUNG wire#powerrail
      Contact( "StageLL0" )
   END_RUNG wire#w1
   // the same network as SCL:
   IF "StageLL6" THEN "PumpVLow_bit" := TRUE; END_IF;
   IF "StageLL7" OR "StageLL0" THEN "PumpVLow_bit" := FALSE; END_IF;
END_REGION

REGION Network 7
   RUNG wire#powerrail
      Contact( "StageLL9" )
      S_Coil( "MFillFinish" )
   END_RUNG
   RUNG wire#powerrail
      Contact( "StageLL13" )
      wire#w1
      R_Coil( "MFillFinish" )
   END_RUNG
   RUNG wire#powerrail
      Contact( "StageLL00" )
   END_RUNG wire#w1
   // the same network as SCL:
   IF "StageLL9" THEN "MFillFinish" := TRUE; END_IF;
   IF "StageLL13" OR "StageLL00" THEN "MFillFinish" := FALSE; END_IF;
END_REGION

REGION Network 8
   RUNG wire#powerrail
      Contact( "StageLL9" )
      wire#w1
      Coil( "MBottleCounterR" )
   END_RUNG
   RUNG wire#powerrail
      I_Contact( "E_stop_bit" )
   END_RUNG wire#w1
   RUNG wire#powerrail
      Contact( "Stop_hmi" )
   END_RUNG wire#w1
   // the same network as SCL:
   "MBottleCounterR" := "StageLL9" OR NOT "E_stop_bit" OR "Stop_hmi";
END_REGION

REGION Network 9
   RUNG wire#powerrail
      Contact( "StageLL10" )
      wire#w1
      Coil( "ProcessFillingTimeR" )
   END_RUNG
   RUNG wire#powerrail
      I_Contact( "E_stop_bit" )
   END_RUNG wire#w1
   RUNG wire#powerrail
      Contact( "Stop_hmi" )
   END_RUNG wire#w1
   // the same network as SCL:
   "ProcessFillingTimeR" := "StageLL10" OR NOT "E_stop_bit" OR "Stop_hmi";
END_REGION

REGION Network 10
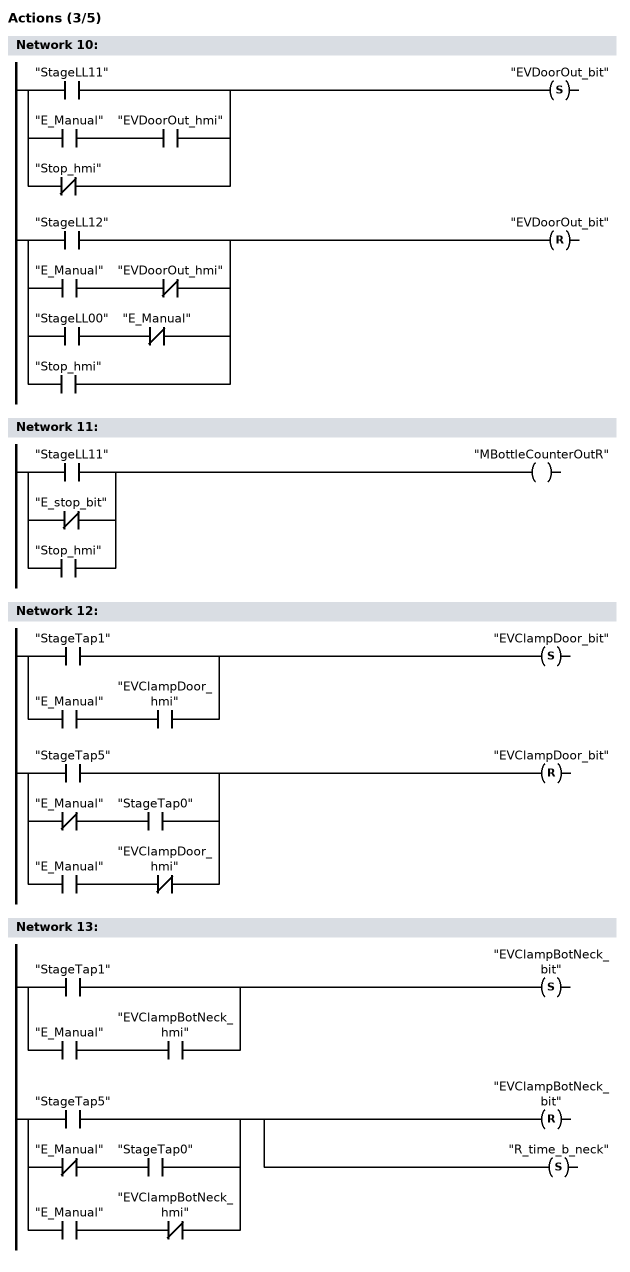
   RUNG wire#powerrail
      Contact( "StageLL11" )
      wire#w1
      S_Coil( "EVDoorOut_bit" )
   END_RUNG
   RUNG wire#powerrail
      Contact( "E_Manual" )
      Contact( "EVDoorOut_hmi" )
   END_RUNG wire#w1
   RUNG wire#powerrail
      I_Contact( "Stop_hmi" )
   END_RUNG wire#w1
   RUNG wire#powerrail
      Contact( "StageLL12" )
      wire#w2
      R_Coil( "EVDoorOut_bit" )
   END_RUNG
   RUNG wire#powerrail
      Contact( "E_Manual" )
      I_Contact( "EVDoorOut_hmi" )
   END_RUNG wire#w2
   RUNG wire#powerrail
      Contact( "StageLL00" )
      I_Contact( "E_Manual" )
   END_RUNG wire#w2
   RUNG wire#powerrail
      Contact( "Stop_hmi" )
   END_RUNG wire#w2
   // the same network as SCL:
   IF "StageLL11" OR ("E_Manual" AND "EVDoorOut_hmi") OR NOT "Stop_hmi" THEN "EVDoorOut_bit" := TRUE; END_IF;
   IF "StageLL12" OR ("E_Manual" AND NOT "EVDoorOut_hmi") OR ("StageLL00" AND NOT "E_Manual") OR "Stop_hmi" THEN
       "EVDoorOut_bit" := FALSE;
   END_IF;
END_REGION

REGION Network 11
   RUNG wire#powerrail
      Contact( "StageLL11" )
      wire#w1
      Coil( "MBottleCounterOutR" )
   END_RUNG
   RUNG wire#powerrail
      I_Contact( "E_stop_bit" )
   END_RUNG wire#w1
   RUNG wire#powerrail
      Contact( "Stop_hmi" )
   END_RUNG wire#w1
   // the same network as SCL:
   "MBottleCounterOutR" := "StageLL11" OR NOT "E_stop_bit" OR "Stop_hmi";
END_REGION

REGION Network 12
   RUNG wire#powerrail
      Contact( "StageTap1" )
      wire#w1
      S_Coil( "EVClampDoor_bit" )
   END_RUNG
   RUNG wire#powerrail
      Contact( "E_Manual" )
      Contact( "EVClampDoor_hmi" )
   END_RUNG wire#w1
   RUNG wire#powerrail
      Contact( "StageTap5" )
      wire#w2
      R_Coil( "EVClampDoor_bit" )
   END_RUNG
   RUNG wire#powerrail
      I_Contact( "E_Manual" )
      Contact( "StageTap0" )
   END_RUNG wire#w2
   RUNG wire#powerrail
      Contact( "E_Manual" )
      I_Contact( "EVClampDoor_hmi" )
   END_RUNG wire#w2
   // the same network as SCL:
   IF "StageTap1" OR ("E_Manual" AND "EVClampDoor_hmi") THEN "EVClampDoor_bit" := TRUE; END_IF;
   IF "StageTap5" OR (NOT "E_Manual" AND "StageTap0") OR ("E_Manual" AND NOT "EVClampDoor_hmi") THEN
       "EVClampDoor_bit" := FALSE;
   END_IF;
END_REGION

REGION Network 13
   RUNG wire#powerrail
      Contact( "StageTap1" )
      wire#w1
      S_Coil( "EVClampBotNeck_bit" )
   END_RUNG
   RUNG wire#powerrail
      Contact( "E_Manual" )
      Contact( "EVClampBotNeck_hmi" )
   END_RUNG wire#w1
   RUNG wire#powerrail
      Contact( "StageTap5" )
      wire#w2
      R_Coil( "EVClampBotNeck_bit" )
   END_RUNG
   RUNG wire#powerrail
      I_Contact( "E_Manual" )
      Contact( "StageTap0" )
   END_RUNG wire#w2
   RUNG wire#powerrail
      Contact( "E_Manual" )
      I_Contact( "EVClampBotNeck_hmi" )
   END_RUNG wire#w2
   RUNG wire#w2
      S_Coil( "R_time_b_neck" )
   END_RUNG
   // the same network as SCL:
   IF "StageTap1" OR ("E_Manual" AND "EVClampBotNeck_hmi") THEN "EVClampBotNeck_bit" := TRUE; END_IF;
   IF "StageTap5" OR (NOT "E_Manual" AND "StageTap0") OR ("E_Manual" AND NOT "EVClampBotNeck_hmi") THEN
       "EVClampBotNeck_bit" := FALSE;
       "R_time_b_neck" := TRUE;
   END_IF;
END_REGION

REGION Network 15
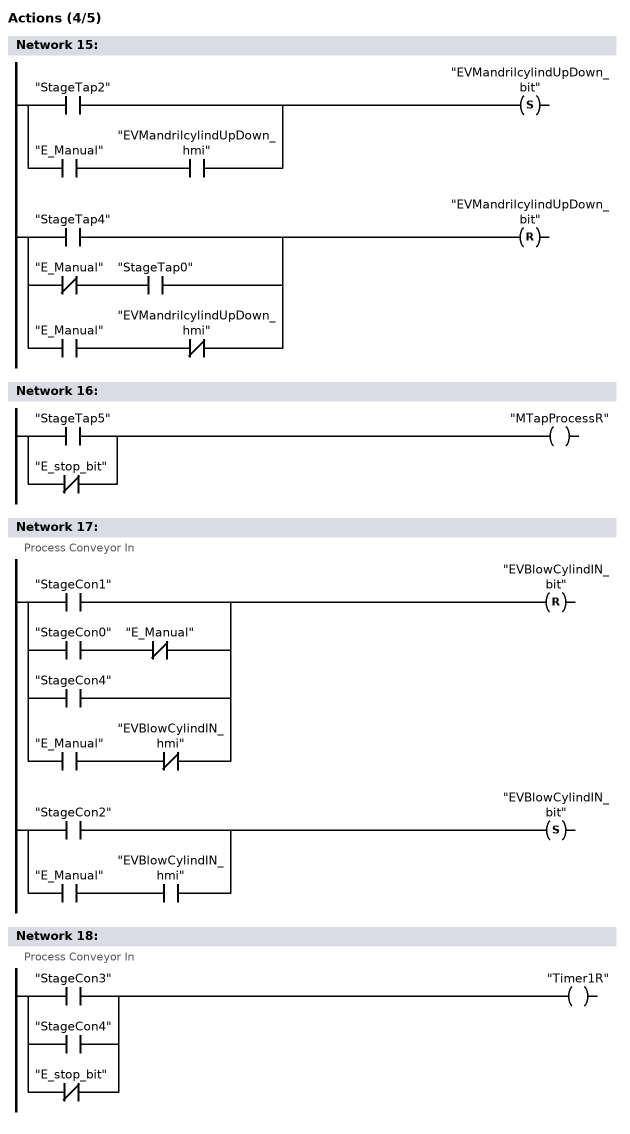
   RUNG wire#powerrail
      Contact( "StageTap2" )
      wire#w1
      S_Coil( "EVMandrilcylindUpDown_bit" )
   END_RUNG
   RUNG wire#powerrail
      Contact( "E_Manual" )
      Contact( "EVMandrilcylindUpDown_hmi" )
   END_RUNG wire#w1
   RUNG wire#powerrail
      Contact( "StageTap4" )
      wire#w2
      R_Coil( "EVMandrilcylindUpDown_bit" )
   END_RUNG
   RUNG wire#powerrail
      I_Contact( "E_Manual" )
      Contact( "StageTap0" )
   END_RUNG wire#w2
   RUNG wire#powerrail
      Contact( "E_Manual" )
      I_Contact( "EVMandrilcylindUpDown_hmi" )
   END_RUNG wire#w2
   // the same network as SCL:
   IF "StageTap2" OR ("E_Manual" AND "EVMandrilcylindUpDown_hmi") THEN
       "EVMandrilcylindUpDown_bit" := TRUE;
   END_IF;
   IF "StageTap4" OR (NOT "E_Manual" AND "StageTap0") OR ("E_Manual" AND NOT "EVMandrilcylindUpDown_hmi") THEN
       "EVMandrilcylindUpDown_bit" := FALSE;
   END_IF;
END_REGION

REGION Network 16
   RUNG wire#powerrail
      Contact( "StageTap5" )
      wire#w1
      Coil( "MTapProcessR" )
   END_RUNG
   RUNG wire#powerrail
      I_Contact( "E_stop_bit" )
   END_RUNG wire#w1
   // the same network as SCL:
   "MTapProcessR" := "StageTap5" OR NOT "E_stop_bit";
END_REGION

REGION Network 17
   // Process Conveyor In
   RUNG wire#powerrail
      Contact( "StageCon1" )
      wire#w1
      R_Coil( "EVBlowCylindIN_bit" )
   END_RUNG
   RUNG wire#powerrail
      Contact( "StageCon0" )
      I_Contact( "E_Manual" )
   END_RUNG wire#w1
   RUNG wire#powerrail
      Contact( "StageCon4" )
   END_RUNG wire#w1
   RUNG wire#powerrail
      Contact( "E_Manual" )
      I_Contact( "EVBlowCylindIN_hmi" )
   END_RUNG wire#w1
   RUNG wire#powerrail
      Contact( "StageCon2" )
      wire#w2
      S_Coil( "EVBlowCylindIN_bit" )
   END_RUNG
   RUNG wire#powerrail
      Contact( "E_Manual" )
      Contact( "EVBlowCylindIN_hmi" )
   END_RUNG wire#w2
   // the same network as SCL:
   IF "StageCon1" OR ("StageCon0" AND NOT "E_Manual") OR "StageCon4" OR ("E_Manual" AND NOT "EVBlowCylindIN_hmi") THEN
       "EVBlowCylindIN_bit" := FALSE;
   END_IF;
   IF "StageCon2" OR ("E_Manual" AND "EVBlowCylindIN_hmi") THEN "EVBlowCylindIN_bit" := TRUE; END_IF;
END_REGION

REGION Network 18
   // Process Conveyor In
   RUNG wire#powerrail
      Contact( "StageCon3" )
      wire#w1
      Coil( "Timer1R" )
   END_RUNG
   RUNG wire#powerrail
      Contact( "StageCon4" )
   END_RUNG wire#w1
   RUNG wire#powerrail
      I_Contact( "E_stop_bit" )
   END_RUNG wire#w1
   // the same network as SCL:
   "Timer1R" := "StageCon3" OR "StageCon4" OR NOT "E_stop_bit";
END_REGION

REGION Network 19
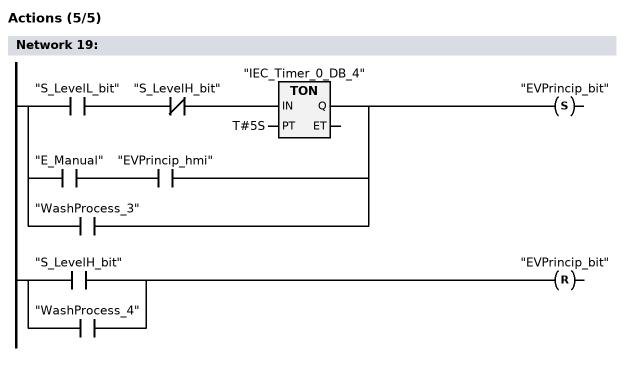
   "IEC_Timer_0_DB_4".TON(IN := "S_LevelL_bit" AND NOT "S_LevelH_bit", PT := T#5S);
   IF "IEC_Timer_0_DB_4".Q OR ("E_Manual" AND "EVPrincip_hmi") OR "WashProcess_3" THEN
       "EVPrincip_bit" := TRUE;
   END_IF;
   IF "S_LevelH_bit" OR "WashProcess_4" THEN "EVPrincip_bit" := FALSE; END_IF;
END_REGION
END_ORGANIZATION_BLOCK

ORGANIZATION_BLOCK "Block_convertion"   // OB127, LAD, ProgramCycle
TITLE = "Main Program Sweep (Cycle)"
{ S7_Optimized_Access := 'TRUE' }
VERSION : 0.1
   VAR_INPUT
      Initial_Call : Bool;   // Initial call of this OB
      Remanence : Bool;   // =True, if remanent data are available
   END_VAR
   VAR_TEMP   // added for the SCL form of the ladder/FBD networks
      _w1 : Bool;
   END_VAR
BEGIN

REGION Network 1
   // Data HMI Delay
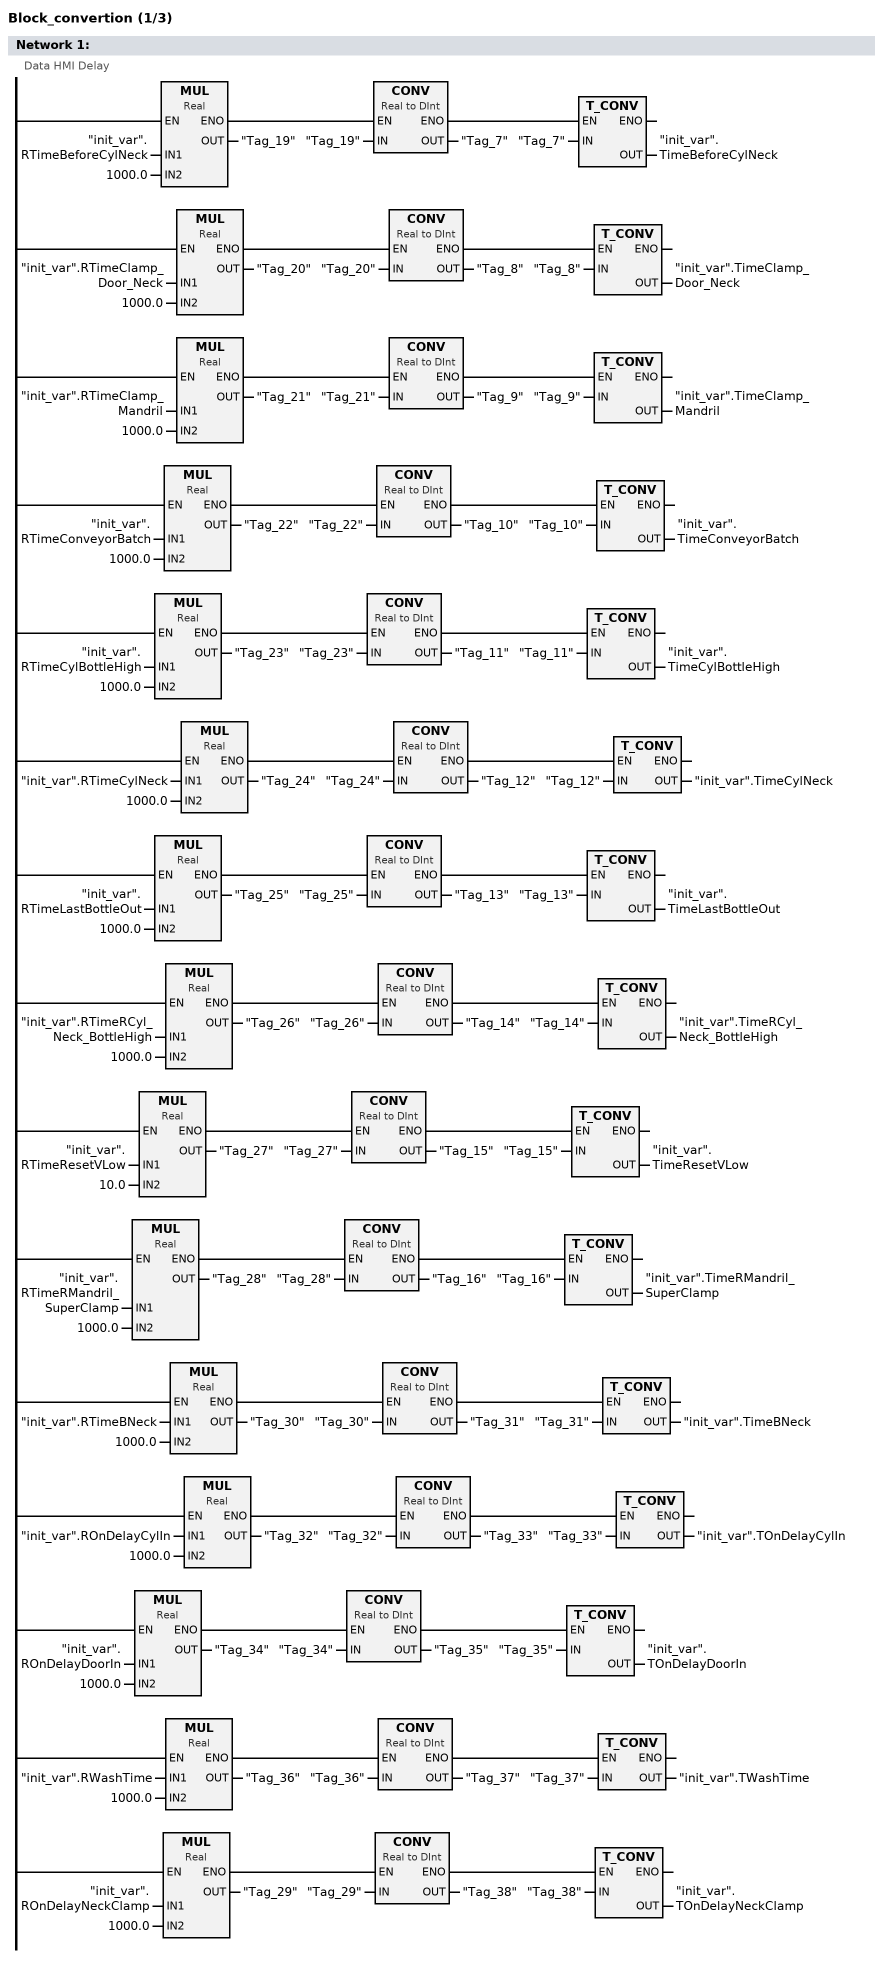
   "Tag_19" := "init_var".RTimeBeforeCylNeck * 1000.0;
   "Tag_7" := REAL_TO_DINT("Tag_19");
   "init_var".TimeBeforeCylNeck := T_CONV(IN := "Tag_7");
   "Tag_20" := "init_var".RTimeClamp_Door_Neck * 1000.0;
   "Tag_8" := REAL_TO_DINT("Tag_20");
   "init_var".TimeClamp_Door_Neck := T_CONV(IN := "Tag_8");
   "Tag_21" := "init_var".RTimeClamp_Mandril * 1000.0;
   "Tag_9" := REAL_TO_DINT("Tag_21");
   "init_var".TimeClamp_Mandril := T_CONV(IN := "Tag_9");
   "Tag_22" := "init_var".RTimeConveyorBatch * 1000.0;
   "Tag_10" := REAL_TO_DINT("Tag_22");
   "init_var".TimeConveyorBatch := T_CONV(IN := "Tag_10");
   "Tag_23" := "init_var".RTimeCylBottleHigh * 1000.0;
   "Tag_11" := REAL_TO_DINT("Tag_23");
   "init_var".TimeCylBottleHigh := T_CONV(IN := "Tag_11");
   "Tag_24" := "init_var".RTimeCylNeck * 1000.0;
   "Tag_12" := REAL_TO_DINT("Tag_24");
   "init_var".TimeCylNeck := T_CONV(IN := "Tag_12");
   "Tag_25" := "init_var".RTimeLastBottleOut * 1000.0;
   "Tag_13" := REAL_TO_DINT("Tag_25");
   "init_var".TimeLastBottleOut := T_CONV(IN := "Tag_13");
   "Tag_26" := "init_var".RTimeRCyl_Neck_BottleHigh * 1000.0;
   "Tag_14" := REAL_TO_DINT("Tag_26");
   "init_var".TimeRCyl_Neck_BottleHigh := T_CONV(IN := "Tag_14");
   "Tag_27" := "init_var".RTimeResetVLow * 10.0;
   "Tag_15" := REAL_TO_DINT("Tag_27");
   "init_var".TimeResetVLow := T_CONV(IN := "Tag_15");
   "Tag_28" := "init_var".RTimeRMandril_SuperClamp * 1000.0;
   "Tag_16" := REAL_TO_DINT("Tag_28");
   "init_var".TimeRMandril_SuperClamp := T_CONV(IN := "Tag_16");
   "Tag_30" := "init_var".RTimeBNeck * 1000.0;
   "Tag_31" := REAL_TO_DINT("Tag_30");
   "init_var".TimeBNeck := T_CONV(IN := "Tag_31");
   "Tag_32" := "init_var".ROnDelayCylIn * 1000.0;
   "Tag_33" := REAL_TO_DINT("Tag_32");
   "init_var".TOnDelayCylIn := T_CONV(IN := "Tag_33");
   "Tag_34" := "init_var".ROnDelayDoorIn * 1000.0;
   "Tag_35" := REAL_TO_DINT("Tag_34");
   "init_var".TOnDelayDoorIn := T_CONV(IN := "Tag_35");
   "Tag_36" := "init_var".RWashTime * 1000.0;
   "Tag_37" := REAL_TO_DINT("Tag_36");
   "init_var".TWashTime := T_CONV(IN := "Tag_37");
   "Tag_29" := "init_var".ROnDelayNeckClamp * 1000.0;
   "Tag_38" := REAL_TO_DINT("Tag_29");
   "init_var".TOnDelayNeckClamp := T_CONV(IN := "Tag_38");
END_REGION

REGION Network 2
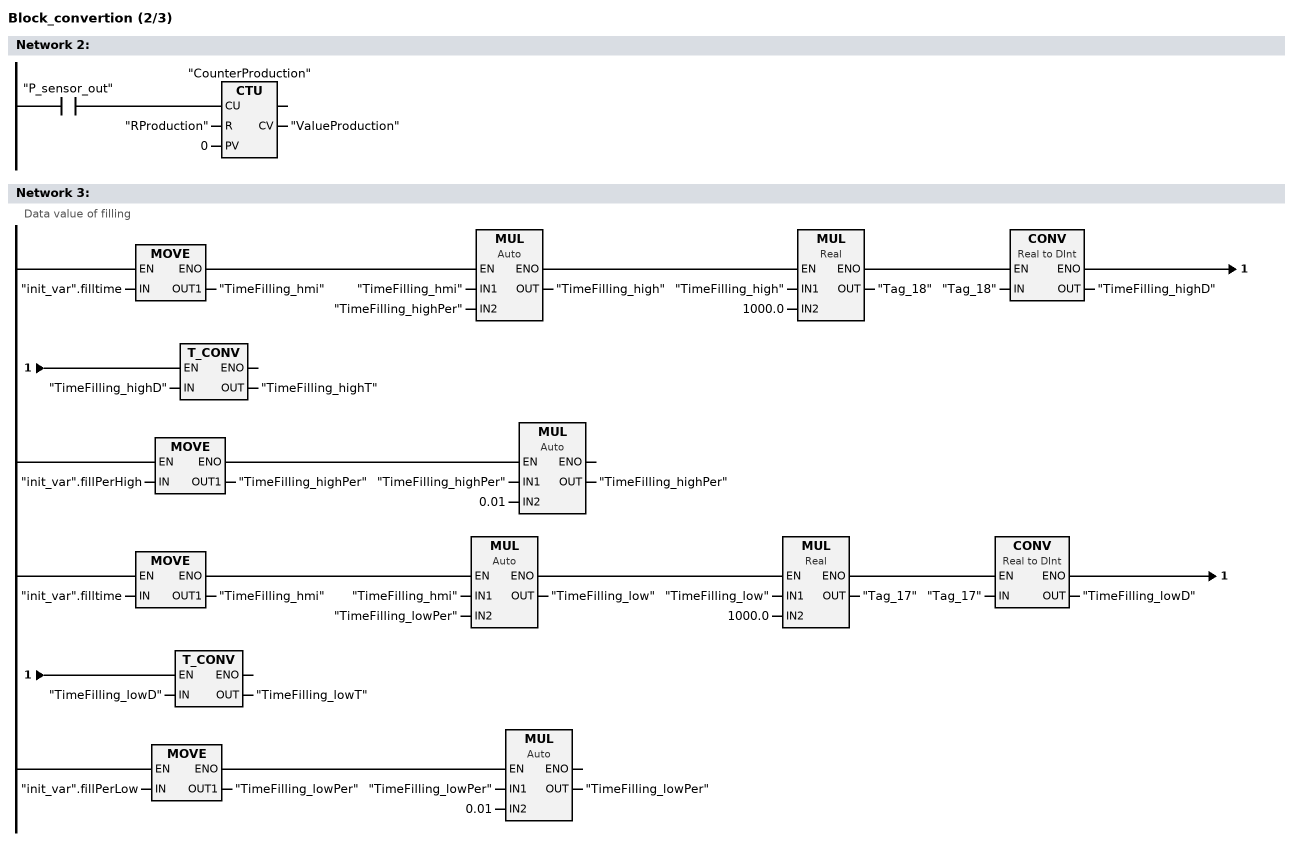
   "CounterProduction".CTU(CU := "P_sensor_out", R := "RProduction", PV := 0, CV => "ValueProduction");
END_REGION

REGION Network 3
   // Data value of filling
   "TimeFilling_hmi" := "init_var".filltime;
   "TimeFilling_high" := "TimeFilling_hmi" * "TimeFilling_highPer";
   "Tag_18" := "TimeFilling_high" * 1000.0;
   "TimeFilling_highD" := REAL_TO_DINT("Tag_18");
   "TimeFilling_highT" := T_CONV(IN := "TimeFilling_highD");
   "TimeFilling_highPer" := "init_var".fillPerHigh;
   "TimeFilling_highPer" := "TimeFilling_highPer" * 0.01;
   "TimeFilling_hmi" := "init_var".filltime;
   "TimeFilling_low" := "TimeFilling_hmi" * "TimeFilling_lowPer";
   "Tag_17" := "TimeFilling_low" * 1000.0;
   "TimeFilling_lowD" := REAL_TO_DINT("Tag_17");
   "TimeFilling_lowT" := T_CONV(IN := "TimeFilling_lowD");
   "TimeFilling_lowPer" := "init_var".fillPerLow;
   "TimeFilling_lowPer" := "TimeFilling_lowPer" * 0.01;
END_REGION

REGION Network 4
   // Production data calculation
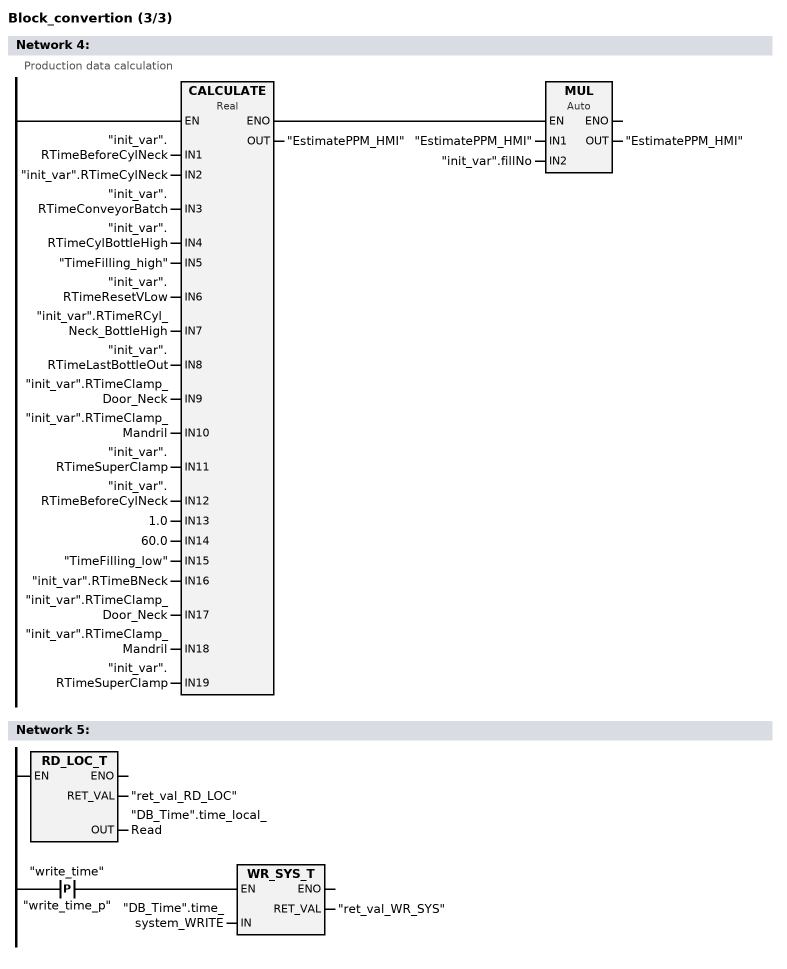
   RUNG wire#powerrail
      { S7_Templates := "SrcType := Real"; S7_Expression := "(IN13*IN14)/(IN1+IN2+IN3+IN4+IN5+IN6+IN7+IN8+IN9+IN10+IN11+IN12+IN15+IN16+IN17+IN18+IN19)" } Calculate(in1 := "init_var".RTimeBeforeCylNeck, in2 := "init_var".RTimeCylNeck, in3 := "init_var".RTimeConveyorBatch, in4 := "init_var".RTimeCylBottleHigh, in5 := "TimeFilling_high", in6 := "init_var".RTimeResetVLow, in7 := "init_var".RTimeRCyl_Neck_BottleHigh, in8 := "init_var".RTimeLastBottleOut, in9 := "init_var".RTimeClamp_Door_Neck, in10 := "init_var".RTimeClamp_Mandril, in11 := "init_var".RTimeSuperClamp, in12 := "init_var".RTimeBeforeCylNeck, in13 := 1.0, in14 := 60.0, in15 := "TimeFilling_low", in16 := "init_var".RTimeBNeck, in17 := "init_var".RTimeClamp_Door_Neck, in18 := "init_var".RTimeClamp_Mandril, in19 := "init_var".RTimeSuperClamp, out => "EstimatePPM_HMI")
      Mul(in1 := "EstimatePPM_HMI", in2 := "init_var".fillNo, out => "EstimatePPM_HMI")
   END_RUNG
   // the same network as SCL:
   "EstimatePPM_HMI" := (1.0*60.0)/("init_var".RTimeBeforeCylNeck+"init_var".RTimeCylNeck+"init_var".RTimeConveyorBatch+"init_var".RTimeCylBottleHigh+"TimeFilling_high"+"init_var".RTimeResetVLow+"init_var".RTimeRCyl_Neck_BottleHigh+"init_var".RTimeLastBottleOut+"init_var".RTimeClamp_Door_Neck+"init_var".RTimeClamp_Mandril+"init_var".RTimeSuperClamp+"init_var".RTimeBeforeCylNeck+"TimeFilling_low"+"init_var".RTimeBNeck+"init_var".RTimeClamp_Door_Neck+"init_var".RTimeClamp_Mandril+"init_var".RTimeSuperClamp);
   "EstimatePPM_HMI" := "EstimatePPM_HMI" * "init_var".fillNo;
END_REGION

REGION Network 5
   "ret_val_RD_LOC" := RD_LOC_T(OUT => "DB_Time".time_local_Read);
   #_w1 := "write_time" AND NOT "write_time_p";   // rising edge of "write_time"
   "write_time_p" := "write_time";
   IF #_w1 THEN "ret_val_WR_SYS" := WR_SYS_T(IN := "DB_Time".time_system_WRITE); END_IF;
END_REGION
END_ORGANIZATION_BLOCK

(* ===== HMI "HMI_RT_2" =====
system functions are stored by id; their names below are inferred from use
connection "HMI_Connection_1": ETHERNET, SMART_S7_1500_OMS
connection "Connection_1": ETHERNET, SMART_S7_1500_OMS

HMI tags "Default tag table"
   "HMI_Tag_1" : UInt AT %DB13.DBW0, 1 s
   "Tag_ScreenNumber" : UInt, internal
   "Start_hmi" : Bool = PLC Start_hmi AT %M11.0, 1 s
   "E_Trans1_hmi" : Bool = PLC E_Trans1_hmi AT %M27.4, 1 s
   "E_Trans2_hmi" : Bool = PLC E_Trans2_hmi AT %M27.5, 1 s
   "MotorTap_hmi" : Bool = PLC E_MotorTap_hmi AT %M27.7, 1 s
   "ACKTransp1_bit" : Bool = PLC ACKTransp1_bit AT %M32.2, 1 s
   "ACKTransp2_bit" : Bool = PLC ACKTransp2_bit AT %M32.3, 1 s
   "ACKTap_bit" : Bool = PLC ACKTap_bit AT %M32.0, 1 s
   "MotorTrans2_bit" : Bool = PLC MotorTrans2_bit AT %M22.1, 1 s
   "init_var_filltime" : Real = PLC init_var.filltime, 1 s
   "M_stop_hmi" : Bool = PLC M_stop_hmi AT %M11.1, 1 s
   "init_var_fillNo" : Int = PLC init_var.fillNo, 1 s
   "EVPrincip_bit" : Bool = PLC EVPrincip_bit AT %M22.2, 1 s
   "PumpVLow_bit" : Bool = PLC PumpVLow_bit AT %M21.4, 1 s
   "ACKPump_bit" : Bool = PLC ACKPump_bit AT %M32.1, 1 s
   "EVCylindBottleHigh_bit" : Bool = PLC EVCylindBottleHigh_bit AT %M28.0, 1 s
   "EVBlowCylindIN_bit" : Bool = PLC EVBlowCylindIN_bit AT %M22.3, 1 s
   "EVClampBotNeck_bit" : Bool = PLC EVClampBotNeck_bit AT %M23.0, 1 s
   "EVDoorIn_bit" : Bool = PLC EVDoorIn_bit AT %M50.1, 1 s
   "EVDoorOut_bit" : Bool = PLC EVDoorOut_bit AT %M22.7, 1 s
   "EVCylindNeck_bit" : Bool = PLC EVCylindNeck_bit AT %M22.5, 1 s
   "EVClampDoor_bit" : Bool = PLC EVClampDoor_bit AT %M23.1, 1 s
   "EVSuperClamp_bit" : Bool = PLC EVSuperClamp_bit AT %M23.2, 1 s
   "EVMandrilcylindUpDown_bit" : Bool = PLC EVMandrilcylindUpDown_bit AT %M22.4, 1 s
   "TapPPM_HMI" : Word = PLC TapPPM_HMI AT %MW6, 1 s
   "init_var_fillPerHigh" : Real = PLC init_var.fillPerHigh, 1 s
   "init_var_fillPerLow" : Real = PLC init_var.fillPerLow, 1 s
   "EstimatePPM_HMI" : Real = PLC EstimatePPM_HMI AT %MD70, 1 s
   "E_Stop" : Bool = PLC E_Stop AT %I0.0, 1 s
   "F_TriggerPump" : Bool = PLC F_TriggerPump AT %I0.1, 1 s
   "ACKPump" : Bool = PLC ACKPump AT %I0.2, 1 s
   "F_TriggerClamp" : Bool = PLC F_TriggerClamp AT %I0.3, 1 s
   "ACKTap" : Bool = PLC ACKTap AT %I0.4, 1 s
   "F_TriggerTransp1" : Bool = PLC F_TriggerTransp1 AT %I0.5, 1 s
   "ACKTransp1" : Bool = PLC ACKTransp1 AT %I0.6, 1 s
   "F_TriggerTransp2" : Bool = PLC F_TriggerTransp2 AT %I0.7, 1 s
   "ACKTransp2" : Bool = PLC ACKTransp2 AT %I1.0, 1 s
   "S_ConvellorClearence_In" : Bool = PLC S_ConvellorClearence_In AT %I1.1, 1 s
   "S_InBottle" : Bool = PLC S_InBottle AT %I1.2, 1 s
   "S_OutBottle" : Bool = PLC S_OutBottle AT %I1.6, 1 s
   "S_LastBottle" : Bool = PLC S_LastBottle AT %I1.4, 1 s
   "S_Bottle_Convellor1" : Bool = PLC S_Bottle_Convellor1 AT %I1.5, 1 s
   "S_LevelH" : Bool = PLC S_LevelH AT %I1.3, 1 s
   "S_LevelL" : Bool = PLC S_LevelL AT %I1.7, 1 s
   "S_BottleTap" : Bool = PLC S_BottleTap AT %I2.0, 1 s
   "S_TranspClamp" : Bool = PLC S_TranspClamp AT %I2.1, 1 s
   "PumpVLow" : Bool = PLC PumpVLow AT %Q0.0, 1 s
   "PumpVHigh" : Bool = PLC PumpVHigh AT %Q0.1, 1 s
   "PumpStop" : Bool = PLC PumpStop AT %Q0.2, 1 s
   "MotorTap" : Bool = PLC MotorTap AT %Q0.3, 1 s
   "MotorTrans1" : Bool = PLC MotorTrans1 AT %Q0.4, 1 s
   "MotorTrans2" : Bool = PLC MotorTrans2 AT %Q0.5, 1 s
   "EVPrincip" : Bool = PLC EVPrincip AT %Q1.6, 1 s
   "EVBlowCylindIN" : Bool = PLC EVBlowCylindIN AT %Q1.7, 1 s
   "EVCylindBottleHigh" : Bool = PLC EVCylindBottleHigh AT %Q2.0, 1 s
   "EVCylindNeck" : Bool = PLC EVCylindNeck AT %Q2.1, 1 s
   "EVDoorIn" : Bool = PLC EVDoorIn AT %Q2.2, 1 s
   "EVDoorOut" : Bool = PLC EVDoorOut AT %Q2.3, 1 s
   "EVClampBotNeck" : Bool = PLC EVClampBotNeck AT %Q2.4, 1 s
   "EVClampDoor" : Bool = PLC EVClampDoor AT %Q2.5, 1 s
   "EVSuperClamp" : Bool = PLC EVSuperClamp AT %Q2.6, 1 s
   "EVMandrilcylindUpDown" : Bool = PLC EVMandrilcylindUpDown AT %Q2.7, 1 s
   "EVCylindBottleHigh_hmi" : Bool = PLC EVCylindBottleHigh_hmi AT %M37.7, 1 s
   "EVCylindNeck_hmi" : Bool = PLC EVCylindNeck_hmi AT %M39.0, 1 s
   "EVBlowCylindIN_hmi" : Bool = PLC EVBlowCylindIN_hmi AT %M37.6, 1 s
   "EVPrincip_hmi" : Bool = PLC EVPrincip_hmi AT %M39.1, 1 s
   "EVDoorOut_hmi" : Bool = PLC EVDoorOut_hmi AT %M39.3, 1 s
   "EVClampBotNeck_hmi" : Bool = PLC EVClampBotNeck_hmi AT %M39.4, 1 s
   "EVClampDoor_hmi" : Bool = PLC EVClampDoor_hmi AT %M39.5, 1 s
   "EVSuperClamp_hmi" : Bool = PLC EVSuperClamp_hmi AT %M50.2, 1 s
   "EVMandrilcylindUpDown_hmi" : Bool = PLC EVMandrilcylindUpDown_hmi AT %M50.3, 1 s
   "PumpVLow_hmi" : Bool = PLC PumpVLow_hmi AT %M37.5, 1 s
   "E_Manual_hmi" : Bool = PLC E_Manual_hmi AT %M31.6, 1 s
   "init_var_TimeBeforeCylNeck" : Time = PLC init_var.TimeBeforeCylNeck, 1 s
   "init_var_TimeCylNeck" : Time = PLC init_var.TimeCylNeck, 1 s
   "init_var_TimeCylBottleHigh" : Time = PLC init_var.TimeCylBottleHigh, 1 s
   "TimeFilling_highT" : Time = PLC TimeFilling_highT AT %MD116, 1 s
   "TimeFilling_lowT" : Time = PLC TimeFilling_lowT AT %MD120, 1 s
   "init_var_TimeResetVLow" : Time = PLC init_var.TimeResetVLow, 1 s
   "EVDoorIn_hmi" : Bool = PLC EVDoorIn_hmi AT %M50.0, 1 s
   "init_var_RTimeBeforeCylNeck" : Real = PLC init_var.RTimeBeforeCylNeck, 1 s
   "init_var_RTimeCylNeck" : Real = PLC init_var.RTimeCylNeck, 1 s
   "init_var_RTimeCylBottleHigh" : Real = PLC init_var.RTimeCylBottleHigh, 1 s
   "init_var_RTimeResetVLow" : Real = PLC init_var.RTimeResetVLow, 1 s
   "init_var_TimeLastBottleOut" : Time = PLC init_var.TimeLastBottleOut, 1 s
   "init_var_RTimeLastBottleOut" : Real = PLC init_var.RTimeLastBottleOut, 1 s
   "TimeFilling_low" : Real = PLC TimeFilling_low AT %MD112, 1 s
   "TimeFilling_high" : Real = PLC TimeFilling_high AT %MD104, 1 s
   "init_var_RTimeClamp_Door_Neck" : Real = PLC init_var.RTimeClamp_Door_Neck, 1 s
   "init_var_RTimeClamp_Mandril" : Real = PLC init_var.RTimeClamp_Mandril, 1 s
   "init_var_TimeBNeck" : Time = PLC init_var.TimeBNeck, 1 s
   "init_var_RTimeBNeck" : Real = PLC init_var.RTimeBNeck, 1 s
   "PumpVHihg_hmi" : Bool = PLC PumpVHihg_hmi AT %M40.2, 1 s
   "init_var_ROnDelayCylIn" : Real = PLC init_var.ROnDelayCylIn, 1 s
   "init_var_TOnDelayDoorIn" : Time = PLC init_var.TOnDelayDoorIn, 1 s
   "init_var_ROnDelayDoorIn" : Real = PLC init_var.ROnDelayDoorIn, 1 s
   "init_var_ROnDelayNeckClamp" : Real = PLC init_var.ROnDelayNeckClamp, 1 s
   "WashProcess_hmi" : Bool = PLC WashProcess_hmi AT %M10.5, 1 s
   "init_var_RWashTime" : Real = PLC init_var.RWashTime, 1 s
   "RProduction" : Bool = PLC RProduction AT %M31.7, 1 s
   "ValueProduction" : DWord = PLC ValueProduction AT %MD272, 1 s
   "init_var_RTimeRCyl_Neck_BottleHigh" : Real = PLC init_var.RTimeRCyl_Neck_BottleHigh, 1 s
   "DB_Time_time_local_Read" : DTL = PLC DB_Time.time_local_Read, 1 s
   "DB_Time_time_system_WRITE" : DTL = PLC DB_Time.time_system_WRITE, 1 s
   "write_time" : Bool = PLC write_time AT %M140.2, 1 s

discrete alarms
   1: 'Alarma Paro de emergencia', class Errors, trigger "HMI_Tag_1" bit 8
   7: 'Disparo de Bomba', class Errors, trigger "HMI_Tag_1" bit 9
   8: 'Disparo del Motor Transportador 1', class Errors, trigger "HMI_Tag_1" bit 10
   9: 'Disparo del Motor Transportador 2', class Errors, trigger "HMI_Tag_1" bit 11
   10: 'Disparo del Motor Taponador', class Errors, trigger "HMI_Tag_1" bit 12
   11: 'Alarmas Activas', class Errors, trigger "HMI_Tag_1" bit 13

Template "Template_1" 320x240
   Button "Shutdown" at 266,202 size 52x37; TextOff 'Text'; PictureOff "ExitRuntime_KTP700_Basic_PN_TR"; Authorization "Programmer"
      on Release: StopRuntime(0)
   Button "Support" at 160,202 size 52x37; TextOff 'Text'; PictureOff "Graphic_4"
      on Release: ActivateScreen("Test", 0)
   Button "Test" at 213,202 size 52x37; TextOff 'Text'; PictureOff "Graphic_2"
      on Release: ActivateScreen("Support", 0)
   Button "Process" at 107,202 size 52x37; TextOff 'Text'; PictureOff "Graphic_3"
      on Release: ActivateScreen("Process", 0)
   Button "Template_Button_4" at 54,202 size 52x37; TextOff 'Text'; PictureOff "AlarmDisplay_KTP700_Basic_PN_TR"
      on Release: ActivateScreen("Alarms", 0)
   Button "Main" at 1,202 size 52x37; TextOff 'Alarms'; PictureOn "AlarmDisplay_KTP600_Basic_color_PN"; PictureOff "NavigateHome_KTP700_Basic_PN_TR"
      on Release: ActivateScreen("Main", 0)
   SymbolicIOField "Symbolic_IO_Field_Screen" at 99,7 size 134x24; TextOff '0'; TextOn '1'; TextList "TextList_ScreenNames"
      on Change: ActivateScreenByNumber("Tag_ScreenNumber", 0)
      ProcessValue <- "Tag_ScreenNumber"
   DateTimeField "HmiScreenItemData" at 235,19 size 85x19
   DateTimeField "HmiScreenItemData_1" at 235,0 size 85x19
   GraphicView "Template_Graphic view_1" at 7,3 size 87x43; Picture "ccn"
   Softkey "Softkey_F1" at 0,0 size 0x0
      on KeyDown: ActivateScreen("Main", 0)
   Softkey "Softkey_F4" at 0,0 size 0x0
      on KeyUp: function_f101fd67("Test")
      on KeyDown: ActivateScreen("Test", 0)
   Softkey "Softkey_F2" at 0,0 size 0x0
      on KeyDown: ActivateScreen("Alarms", 0)
   Softkey "Softkey_F3" at 0,0 size 0x0
      on KeyDown: ActivateScreen("Process", 0)
   Softkey "Softkey_F6" at 0,0 size 0x0
      on KeyDown: function_ee5b8808("Shutdown"); function_f101fd67("Shutdown")
   Softkey "Softkey_F5" at 0,0 size 0x0
      on KeyUp: function_f101fd67("Support")
      on KeyDown: ActivateScreen("Support", 0)

screen "Main" 320x240, template "Template_1"
   on GenerateScreen: SetTag("Tag_ScreenNumber", 1)
   GraphicView "Graphic view_1" at 1,52 size 230x82; Picture "LogoHorizontal-e1441054646412"
   TextField "Text field_3" at 5,154 size 65x18; Text 'Llenadora'
   TextField "Text field_1" at 90,154 size 52x18; Text 'Norland'
   TextField "Text field_2" at 5,174 size 48x18; Text 'Codigo'
   TextField "Text field_4" at 91,174 size 81x18; Text 'BF5000 XLT'
   TextField "Text field_5" at 182,106 size 66x18; Text 'GPM Real'
   IOField "I/O field_1" at 250,97 size 63x26; FormatPattern 9999
      ProcessValue <- "TapPPM_HMI"
   IOField "I/O field_2" at 249,130 size 63x26; FormatPattern 9999
      ProcessValue <- "EstimatePPM_HMI"
   TextField "Text field_6" at 152,138 size 94x18; Text 'GPM Calculado'
   IOField "I/O field_3" at 178,175 size 134x26; FormatPattern 9999999999
      ProcessValue <- "ValueProduction"
   TextField "Text field_7" at 200,157 size 73x18; Text 'Producción'

screen "Alarms" 320x240, template "Template_1"
   on GenerateScreen: SetTag("Tag_ScreenNumber", 2)
   AlarmView "Alarm view_1" at 12,43 size 298x151

screen "Process" 320x240, template "Template_1"
   on GenerateScreen: SetTag("Tag_ScreenNumber", 3)
   Button "HmiScreenItemData_4" at 23,67 size 72x26; TextOn 'SIMATIC PLC system diagnostics'; TextOff 'Transp 1'; PictureOn "Navigates to SIMATIC PLC system diagnostics for HMI_1"; PictureOff "Navigates to SIMATIC PLC system diagnostics for HMI_1"
      on Press: InvertBit("E_Trans1_hmi")
   TextField "Text field_3" at 30,42 size 67x17; Text 'Motores'
   Button "HmiScreenItemData_1" at 23,99 size 72x26; TextOn 'SIMATIC PLC system diagnostics'; TextOff 'Transp 2'; PictureOn "Navigates to SIMATIC PLC system diagnostics for HMI_1"; PictureOff "Navigates to SIMATIC PLC system diagnostics for HMI_1"
      on Press: InvertBit("E_Trans2_hmi")
   Button "HmiScreenItemData_2" at 23,132 size 72x26; TextOn 'SIMATIC PLC system diagnostics'; TextOff 'Motor Tap'; PictureOn "Navigates to SIMATIC PLC system diagnostics for HMI_1"; PictureOff "Navigates to SIMATIC PLC system diagnostics for HMI_1"
      on Press: InvertBit("MotorTap_hmi")
   Rectangle "Rectangle_1" at 95,67 size 12x27
      Appearance <- "E_Trans1_hmi"
   Rectangle "Rectangle_2" at 95,99 size 12x27
      Appearance <- "E_Trans2_hmi"
   Rectangle "Rectangle_3" at 95,132 size 12x27
      Appearance <- "MotorTap_hmi"
   IOField "I/O field_1" at 131,78 size 63x26; FormatPattern 99.9
      ProcessValue <- "init_var_filltime"
   TextField "Text field_1" at 126,42 size 190x17; Text 'Parametros de Llenado'
   TextField "Text field_2" at 194,80 size 15x22; Text 'S'
   TextField "Text field_4" at 239,62 size 57x17; Text '% V. Alta'
   IOField "I/O field_2" at 236,78 size 63x26; FormatPattern 99.9
      ProcessValue <- "init_var_fillPerHigh"
   TextField "Text field_5" at 238,114 size 59x17; Text '% V. Baja'
   IOField "I/O field_3" at 236,132 size 64x26; FormatPattern 99.9
      ProcessValue <- "init_var_fillPerLow"
   Button "Button_1" at 123,168 size 96x32; TextOff 'Start'
      on Press: SetBit("Start_hmi")
      on Release: ResetBit("Start_hmi")
   Button "Button_2" at 230,168 size 82x32; TextOff 'Stop'
      on Press: SetBit("M_stop_hmi")
      Appearance <- "M_stop_hmi"
      on Release: ResetBit("M_stop_hmi")
   TextField "Text field_6" at 141,63 size 44x15; Text 'Tiempo'
   IOField "I/O field_4" at 131,132 size 63x26; FormatPattern 99
      ProcessValue <- "init_var_fillNo"
   TextField "Text field_7" at 139,115 size 47x15; Text 'Botellas'
   Button "Button_3" at 17,168 size 96x32; TextOff 'P. Avanzado'
      on Release: ActivateScreen("Process_stage", 0)

screen "Support" 320x240, template "Template_1"
   on GenerateScreen: SetTag("Tag_ScreenNumber", 5)
   GraphicView "Graphic view_1" at 109,51 size 170x105; Picture "Servicios-de-Consultorias-e-Ingenieria"
   TextField "Text field_1" at 107,153 size 175x16; Text 'contacto info@scisa.com.ni'
   Button "HmiScreenItemData" at 8,57 size 61x24; TextOn 'Online'; TextOff 'Online'
      on Release: function_bb44b551(0)
   Button "HmiScreenItemData_1" at 8,81 size 61x24; TextOn 'Offline'; TextOff 'Offline'
      on Release: function_bb44b551(1)
   Button "HmiScreenItemData_2" at 8,105 size 61x24; TextOn 'Transfer'; TextOff 'Transfer'
      on Release: function_bb44b551(2)
   Button "HmiScreenItemData_3" at 8,129 size 61x24; TextOn 'Toggle language'; TextOff 'Toggle language'
      on Release: function_fb9197e8(-1)
   Button "HmiScreenItemData_4" at 8,153 size 61x24; TextOn 'Toggle language'; TextOff 'Bits PLC'
      on Release: ActivateScreen("DiagnosticIN", 0)
   Button "HmiScreenItemData_5" at 8,178 size 61x24; TextOn 'Toggle language'; TextOff 'Reset C.P.'
      on Release: ResetBit("RProduction")
      on Press: SetBit("RProduction")
   TextField "Text field_2" at 99,169 size 46x14; Text 'Local time'
   IOField "I/O field_2" at 71,180 size 94x21; FormatPattern 9999999999999999999999999999999999999999
      ProcessValue <- "DB_Time_time_local_Read"
   TextField "Text field_3" at 193,169 size 40x14; Text 'Set Time'
   IOField "I/O field_1" at 165,180 size 94x21; FormatPattern 9999999999999999999999999999999999999999
      ProcessValue <- "DB_Time_time_system_WRITE"
   Button "HmiScreenItemData_6" at 259,179 size 60x21; TextOn 'Online'; TextOff 'Set time'
      on Click: SetBit("write_time")
      on Release: ResetBit("write_time")

screen "Test" 320x240, template "Template_1"
   on GenerateScreen: SetTag("Tag_ScreenNumber", 4)
   TextField "Text field_3" at 26,32 size 52x17; Text 'Motores'
   Button "HmiScreenItemData_2" at 9,108 size 70x26; TextOn 'SIMATIC PLC system diagnostics'; TextOff 'Motor Tap'; PictureOn "Navigates to SIMATIC PLC system diagnostics for HMI_1"; PictureOff "Navigates to SIMATIC PLC system diagnostics for HMI_1"
      on Press: InvertBit("MotorTap_hmi")
   Rectangle "Rectangle_1" at 80,51 size 12x27
      Appearance <- "E_Trans1_hmi"
   Rectangle "Rectangle_2" at 80,80 size 12x27
      Appearance <- "E_Trans2_hmi"
   Rectangle "Rectangle_3" at 80,108 size 12x27
      Appearance <- "MotorTap_hmi"
   Button "HmiScreenItemData_3" at 119,51 size 68x26; TextOn 'SIMATIC PLC system diagnostics'; TextOff 'Aliment.'; PictureOn "Navigates to SIMATIC PLC system diagnostics for HMI_1"; PictureOff "Navigates to SIMATIC PLC system diagnostics for HMI_1"
      on Press: InvertBit("EVBlowCylindIN_hmi")
   Rectangle "Rectangle_4" at 188,51 size 12x27
      Appearance <- "EVBlowCylindIN_hmi"
   Button "HmiScreenItemData_4" at 9,51 size 70x26; TextOn 'SIMATIC PLC system diagnostics'; TextOff 'Transp 1'; PictureOn "Navigates to SIMATIC PLC system diagnostics for HMI_1"; PictureOff "Navigates to SIMATIC PLC system diagnostics for HMI_1"
      on Press: InvertBit("E_Trans1_hmi")
   Button "HmiScreenItemData_1" at 9,80 size 70x26; TextOn 'SIMATIC PLC system diagnostics'; TextOff 'Transp 2'; PictureOn "Navigates to SIMATIC PLC system diagnostics for HMI_1"; PictureOff "Navigates to SIMATIC PLC system diagnostics for HMI_1"
      on Press: InvertBit("E_Trans2_hmi")
   Button "HmiScreenItemData_5" at 9,137 size 70x26; TextOn 'SIMATIC PLC system diagnostics'; TextOff 'Bomba'; PictureOn "Navigates to SIMATIC PLC system diagnostics for HMI_1"; PictureOff "Navigates to SIMATIC PLC system diagnostics for HMI_1"
      on Press: InvertBit("PumpVHihg_hmi")
   Rectangle "Rectangle_5" at 80,137 size 12x27
      Appearance <- "PumpVHihg_hmi"
   Button "HmiScreenItemData_6" at 119,80 size 68x26; TextOn 'SIMATIC PLC system diagnostics'; TextOff 'Valvulas'; PictureOn "Navigates to SIMATIC PLC system diagnostics for HMI_1"; PictureOff "Navigates to SIMATIC PLC system diagnostics for HMI_1"
      on Press: InvertBit("EVCylindBottleHigh_hmi")
   Rectangle "Rectangle_6" at 188,80 size 12x27
      Appearance <- "EVCylindBottleHigh_hmi"
   Button "HmiScreenItemData_7" at 119,108 size 68x26; TextOn 'SIMATIC PLC system diagnostics'; TextOff 'Cuello'; PictureOn "Navigates to SIMATIC PLC system diagnostics for HMI_1"; PictureOff "Navigates to SIMATIC PLC system diagnostics for HMI_1"
      on Press: InvertBit("EVCylindNeck_hmi")
   Rectangle "Rectangle_7" at 188,108 size 12x27
      Appearance <- "EVCylindNeck_hmi"
   Button "HmiScreenItemData_8" at 119,137 size 68x26; TextOn 'SIMATIC PLC system diagnostics'; TextOff 'Nivel'; PictureOn "Navigates to SIMATIC PLC system diagnostics for HMI_1"; PictureOff "Navigates to SIMATIC PLC system diagnostics for HMI_1"
      on Press: InvertBit("EVPrincip_hmi")
   Rectangle "Rectangle_8" at 188,137 size 12x27
      Appearance <- "EVPrincip_hmi"
   Button "HmiScreenItemData_9" at 227,51 size 68x26; TextOn 'SIMATIC PLC system diagnostics'; TextOff 'Entrada'; PictureOn "Navigates to SIMATIC PLC system diagnostics for HMI_1"; PictureOff "Navigates to SIMATIC PLC system diagnostics for HMI_1"
      on Press: InvertBit("EVDoorIn_hmi")
   Rectangle "Rectangle_9" at 296,51 size 12x27
      Appearance <- "EVDoorIn_hmi"
   TextField "Text field_1" at 149,33 size 94x17; Text 'Electrovalvulas'
   Button "HmiScreenItemData_10" at 227,80 size 68x26; TextOn 'SIMATIC PLC system diagnostics'; TextOff 'Salida'; PictureOn "Navigates to SIMATIC PLC system diagnostics for HMI_1"; PictureOff "Navigates to SIMATIC PLC system diagnostics for HMI_1"
      on Press: InvertBit("EVDoorOut_hmi")
   Rectangle "Rectangle_10" at 296,80 size 12x26
      Appearance <- "EVDoorOut_bit"
   Button "HmiScreenItemData_11" at 227,108 size 68x26; TextOn 'SIMATIC PLC system diagnostics'; TextOff 'TapCuello'; PictureOn "Navigates to SIMATIC PLC system diagnostics for HMI_1"; PictureOff "Navigates to SIMATIC PLC system diagnostics for HMI_1"
      on Press: InvertBit("EVClampBotNeck_hmi")
   Rectangle "Rectangle_11" at 296,108 size 12x27
      Appearance <- "EVClampBotNeck_bit"
   Rectangle "Rectangle_12" at 296,137 size 12x26
      Appearance <- "EVClampDoor_bit"
   Button "HmiScreenItemData_12" at 227,137 size 68x26; TextOn 'SIMATIC PLC system diagnostics'; TextOff 'TapSalida'; PictureOn "Navigates to SIMATIC PLC system diagnostics for HMI_1"; PictureOff "Navigates to SIMATIC PLC system diagnostics for HMI_1"
      on Press: InvertBit("EVClampDoor_hmi")
   Button "HmiScreenItemData_14" at 227,165 size 68x26; TextOn 'SIMATIC PLC system diagnostics'; TextOff 'Taponar'; PictureOn "Navigates to SIMATIC PLC system diagnostics for HMI_1"; PictureOff "Navigates to SIMATIC PLC system diagnostics for HMI_1"
      on Press: InvertBit("EVMandrilcylindUpDown_hmi")
   Rectangle "Rectangle_14" at 296,165 size 12x27
      Appearance <- "EVMandrilcylindUpDown_bit"
   Button "HmiScreenItemData_15" at 4,168 size 90x34; TextOn 'SIMATIC PLC system diagnostics'; TextOff 'Manual'; PictureOn "Navigates to SIMATIC PLC system diagnostics for HMI_1"; PictureOff "Navigates to SIMATIC PLC system diagnostics for HMI_1"
      on Press: InvertBit("E_Manual_hmi")
      Appearance <- "E_Manual_hmi"
   Button "HmiScreenItemData_13" at 100,176 size 67x24; TextOn 'SIMATIC PLC system diagnostics'; TextOff 'Enjuague'; PictureOn "Navigates to SIMATIC PLC system diagnostics for HMI_1"; PictureOff "Navigates to SIMATIC PLC system diagnostics for HMI_1"
      on Press: SetBit("WashProcess_hmi")
      on Release: ResetBit("WashProcess_hmi")
      Appearance <- "WashProcess_hmi"
   IOField "I/O field_12" at 169,176 size 54x25; FormatPattern 999.9
      ProcessValue <- "init_var_RWashTime"

screen "DiagnosticIN" 320x240, template "Template_1"
   Circle "Circle_1" at 13,57 size 16x16
      Appearance <- "E_Stop"
   TextField "Text field_6" at 31,57 size 24x15; Text 'I0.0'
   Circle "Circle_2" at 13,74 size 16x16
      Appearance <- "F_TriggerPump"
   TextField "Text field_1" at 31,74 size 24x15; Text 'I0.1'
   Circle "Circle_3" at 13,91 size 16x16
      Appearance <- "ACKPump"
   TextField "Text field_2" at 31,91 size 24x15; Text 'I0.2'
   Circle "Circle_4" at 13,108 size 16x16
      Appearance <- "F_TriggerClamp"
   TextField "Text field_3" at 31,108 size 24x15; Text 'I0.3'
   Circle "Circle_5" at 13,125 size 16x16
      Appearance <- "ACKTap"
   TextField "Text field_4" at 31,125 size 24x15; Text 'I0.4'
   Circle "Circle_6" at 13,142 size 16x16
      Appearance <- "F_TriggerTransp1"
   TextField "Text field_5" at 31,142 size 24x15; Text 'I0.5'
   Circle "Circle_7" at 13,159 size 16x16
      Appearance <- "ACKTransp1"
   TextField "Text field_7" at 31,159 size 24x15; Text 'I0.6'
   Circle "Circle_8" at 13,176 size 16x16
      Appearance <- "F_TriggerTransp2"
   TextField "Text field_8" at 31,176 size 24x15; Text 'I0.7'
   Circle "Circle_9" at 57,58 size 16x16
      Appearance <- "ACKTransp2"
   TextField "Text field_9" at 75,58 size 24x15; Text 'I1.0'
   Circle "Circle_10" at 57,75 size 16x16
      Appearance <- "S_ConvellorClearence_In"
   TextField "Text field_10" at 75,75 size 24x15; Text 'I1.1'
   Circle "Circle_11" at 57,92 size 16x16
      Appearance <- "S_InBottle"
   TextField "Text field_11" at 75,92 size 24x15; Text 'I1.2'
   Circle "Circle_12" at 57,109 size 16x16
      Appearance <- "S_OutBottle"
   TextField "Text field_12" at 75,109 size 24x15; Text 'I1.3'
   Circle "Circle_13" at 57,126 size 16x16
      Appearance <- "S_LastBottle"
   TextField "Text field_13" at 75,126 size 24x15; Text 'I1.4'
   Circle "Circle_14" at 57,143 size 16x16
      Appearance <- "S_Bottle_Convellor1"
   TextField "Text field_14" at 75,143 size 24x15; Text 'I1.5'
   Circle "Circle_15" at 57,160 size 16x16
      Appearance <- "S_LevelH"
   TextField "Text field_15" at 75,160 size 24x15; Text 'I1.6'
   Circle "Circle_16" at 57,177 size 16x16
      Appearance <- "S_LevelL"
   TextField "Text field_16" at 75,177 size 24x15; Text 'I1.7'
   Circle "Circle_17" at 101,59 size 16x16
      Appearance <- "S_BottleTap"
   TextField "Text field_17" at 119,59 size 24x15; Text 'I2.0'
   Circle "Circle_18" at 101,76 size 16x16
      Appearance <- "S_TranspClamp"
   TextField "Text field_18" at 119,76 size 24x15; Text 'I2.1'
   Circle "Circle_19" at 101,93 size 16x16
      Appearance <- "E_Stop"
   TextField "Text field_19" at 119,93 size 24x15; Text '̶I̶̶2̶̶.̶̶2̶'
   Circle "Circle_20" at 101,110 size 16x16
      Appearance <- "E_Stop"
   TextField "Text field_20" at 119,110 size 24x15; Text 'I̶̶2̶̶.̶̶3̶'
   Circle "Circle_21" at 101,127 size 16x16
      Appearance <- "E_Stop"
   TextField "Text field_21" at 119,127 size 24x15; Text 'I̶̶2̶̶.̶̶4̶'
   Circle "Circle_22" at 101,144 size 16x16
      Appearance <- "E_Stop"
   TextField "Text field_22" at 119,144 size 24x15; Text 'I̶̶2̶̶.̶̶5̶'
   Circle "Circle_23" at 101,161 size 16x16
      Appearance <- "E_Stop"
   TextField "Text field_23" at 119,161 size 24x15; Text 'I̶̶2̶̶.̶̶6̶'
   Circle "Circle_24" at 101,178 size 16x16
      Appearance <- "E_Stop"
   TextField "Text field_24" at 119,178 size 24x15; Text 'I̶̶2̶̶.̶̶7̶'
   TextField "Text field_25" at 53,41 size 39x15; Text 'Inputs'
   Circle "Circle_25" at 163,59 size 16x16
      Appearance <- "PumpVLow"
   TextField "Text field_26" at 181,59 size 27x15; Text 'Q0.0'
   Circle "Circle_26" at 163,76 size 16x16
      Appearance <- "PumpVHigh"
   TextField "Text field_27" at 181,76 size 27x15; Text 'Q0.1'
   Circle "Circle_27" at 163,93 size 16x16
      Appearance <- "PumpStop"
   TextField "Text field_28" at 181,93 size 27x15; Text 'Q0.2'
   Circle "Circle_28" at 163,110 size 16x16
      Appearance <- "MotorTap"
   TextField "Text field_29" at 181,110 size 27x15; Text 'Q0.3'
   Circle "Circle_29" at 163,127 size 16x16
      Appearance <- "MotorTrans1"
   TextField "Text field_30" at 181,127 size 27x15; Text 'Q0.4'
   Circle "Circle_30" at 163,144 size 16x16
      Appearance <- "MotorTrans2"
   TextField "Text field_31" at 181,144 size 27x15; Text 'Q0.5'
   Circle "Circle_31" at 163,161 size 16x16
      Appearance <- "E_Stop"
   TextField "Text field_32" at 181,161 size 27x15; Text 'Q̶̶0̶̶.̶̶6̶'
   Circle "Circle_32" at 163,178 size 16x16
      Appearance <- "E_Stop"
   TextField "Text field_33" at 181,178 size 27x15; Text 'Q̶̶0̶̶.̶̶7̶'
   Circle "Circle_33" at 209,60 size 16x16
      Appearance <- "E_Stop"
   TextField "Text field_34" at 227,60 size 27x15; Text 'Q̶̶1̶̶.̶̶0̶'
   Circle "Circle_34" at 209,77 size 16x16
      Appearance <- "E_Stop"
   TextField "Text field_35" at 227,77 size 27x15; Text 'Q̶̶1̶̶.̶̶1̶'
   Circle "Circle_35" at 209,94 size 16x16
      Appearance <- "E_Stop"
   TextField "Text field_36" at 227,94 size 27x15; Text 'Q̶̶1̶̶.̶̶2̶'
   Circle "Circle_36" at 209,111 size 16x16
      Appearance <- "E_Stop"
   TextField "Text field_37" at 227,111 size 27x15; Text '̶Q̶̶1̶̶.̶̶3̶'
   Circle "Circle_37" at 209,128 size 16x16
      Appearance <- "E_Stop"
   TextField "Text field_38" at 227,128 size 27x15; Text 'Q̶̶1̶̶.̶̶4̶'
   Circle "Circle_38" at 209,145 size 16x16
      Appearance <- "E_Stop"
   TextField "Text field_39" at 227,145 size 27x15; Text 'Q̶̶1̶̶.̶̶5̶'
   Circle "Circle_39" at 209,162 size 16x16
      Appearance <- "EVPrincip"
   TextField "Text field_40" at 227,162 size 27x15; Text 'Q1.6'
   Circle "Circle_40" at 209,179 size 16x16
      Appearance <- "EVBlowCylindIN"
   TextField "Text field_41" at 227,179 size 27x15; Text 'Q1.7'
   Circle "Circle_41" at 255,61 size 16x16
      Appearance <- "EVCylindBottleHigh"
   TextField "Text field_42" at 273,61 size 27x15; Text 'Q2.0'
   Circle "Circle_42" at 255,78 size 16x16
      Appearance <- "EVCylindNeck"
   TextField "Text field_43" at 273,78 size 27x15; Text 'Q2.1'
   Circle "Circle_43" at 255,95 size 16x16
      Appearance <- "EVDoorIn"
   TextField "Text field_44" at 273,95 size 27x15; Text 'Q2.2'
   Circle "Circle_44" at 255,112 size 16x16
      Appearance <- "EVDoorOut"
   TextField "Text field_45" at 273,112 size 27x15; Text 'Q2.3'
   Circle "Circle_45" at 255,129 size 16x16
      Appearance <- "EVClampBotNeck"
   TextField "Text field_46" at 273,129 size 27x15; Text 'Q2.4'
   Circle "Circle_46" at 255,146 size 16x16
      Appearance <- "EVClampDoor"
   TextField "Text field_47" at 273,146 size 27x15; Text 'Q2.5'
   Circle "Circle_47" at 255,163 size 16x16
      Appearance <- "EVSuperClamp"
   TextField "Text field_48" at 273,163 size 27x15; Text 'Q2.6'
   TextField "Text field_49" at 273,180 size 27x15; Text 'Q2.7'
   TextField "Text field_50" at 207,43 size 47x15; Text 'Outputs'
   Circle "Circle_48" at 255,180 size 16x16
      Appearance <- "EVMandrilcylindUpDown"

screen "Process_stage" 320x240, template "Template_1"
   on GenerateScreen: SetTag("Tag_ScreenNumber", 3)
   TextField "Text field_1" at 91,39 size 139x17; Text 'Parametros de Llenado'
   IOField "I/O field_1" at 19,143 size 52x20; FormatPattern 9.99
      ProcessValue <- "init_var_RTimeBeforeCylNeck"
   TextField "Text field_2" at 70,144 size 13x18; Text 'S'
   TextField "Text field_5" at 20,128 size 50x13; Text 'TD Cuello'
   IOField "I/O field_2" at 19,180 size 52x20; FormatPattern 9.99
      ProcessValue <- "init_var_RTimeCylNeck"
   TextField "Text field_7" at 70,181 size 13x18; Text 'S'
   TextField "Text field_8" at 15,165 size 61x13; Text 'TD Valvulas'
   IOField "I/O field_3" at 90,70 size 52x20; FormatPattern 9.99
      ProcessValue <- "init_var_RTimeCylBottleHigh"
   TextField "Text field_9" at 142,71 size 13x18; Text 'S'
   TextField "Text field_10" at 88,56 size 62x13; Text 'TD Bomba'
   IOField "I/O field_4" at 90,107 size 52x20; FormatPattern 9.99
      ProcessValue <- "TimeFilling_high"
   TextField "Text field_11" at 142,108 size 13x18; Text 'S'
   TextField "Text field_12" at 94,92 size 45x13; Text 'V. Alto'
   IOField "I/O field_5" at 90,143 size 52x20; FormatPattern 9.99
      ProcessValue <- "TimeFilling_low"
   TextField "Text field_4" at 143,144 size 13x18; Text 'S'
   TextField "Text field_6" at 92,128 size 44x13; Text 'V. Baja'
   IOField "I/O field_6" at 90,180 size 52x20; FormatPattern 9.99
      ProcessValue <- "init_var_RTimeResetVLow"
   TextField "Text field_13" at 142,181 size 13x18; Text 'S'
   TextField "Text field_14" at 81,165 size 80x13; Text 'TD R. Valvulas'
   IOField "I/O field_7" at 165,107 size 52x20; FormatPattern 9.99
      ProcessValue <- "init_var_RTimeLastBottleOut"
   TextField "Text field_15" at 217,108 size 13x18; Text 'S'
   TextField "Text field_16" at 159,92 size 58x13; Text 'TD Salida'
   IOField "I/O field_8" at 165,180 size 52x20; FormatPattern 9.99
      ProcessValue <- "init_var_RTimeClamp_Door_Neck"
   TextField "Text field_17" at 219,181 size 13x18; Text 'S'
   TextField "Text field_18" at 171,165 size 41x13; Text 'TD Tap'
   IOField "I/O field_9" at 242,70 size 52x20; FormatPattern 9.99
      ProcessValue <- "init_var_RTimeClamp_Mandril"
   TextField "Text field_19" at 296,71 size 13x18; Text 'S'
   TextField "Text field_20" at 258,55 size 21x13; Text 'Tap'
   IOField "I/O field_10" at 165,143 size 52x20; FormatPattern 9.99
      ProcessValue <- "init_var_RTimeBNeck"
   TextField "Text field_21" at 220,144 size 13x18; Text 'S'
   TextField "Text field_22" at 156,129 size 75x13; Text 'TD Cuello Tap'
   IOField "I/O field_11" at 242,107 size 52x20; FormatPattern 9.99
      ProcessValue <- "init_var_ROnDelayNeckClamp"
   TextField "Text field_23" at 298,108 size 13x18; Text 'S'
   TextField "Text field_24" at 234,92 size 74x13; Text 'TD Salida Tap'
   IOField "I/O field_12" at 19,70 size 52x20; FormatPattern 9.99
      ProcessValue <- "init_var_ROnDelayCylIn"
   TextField "Text field_25" at 70,71 size 13x18; Text 'S'
   TextField "Text field_26" at 13,56 size 67x13; Text 'Alimentador'
   IOField "I/O field_13" at 19,107 size 52x20; FormatPattern 9.99
      ProcessValue <- "init_var_ROnDelayDoorIn"
   TextField "Text field_3" at 70,108 size 13x18; Text 'S'
   TextField "Text field_27" at 16,92 size 61x13; Text 'TD Entrada'
   IOField "I/O field_14" at 165,70 size 52x20; FormatPattern 9.99
      ProcessValue <- "init_var_RTimeRCyl_Neck_BottleHigh"
   TextField "Text field_28" at 218,71 size 13x18; Text 'S'
   TextField "Text field_29" at 157,56 size 68x13; Text 'TD Reset LL'
*)